	                            //table name parts:
	                            #tempTableNameParts := BYTE_TO_USINT(IN := #tdsTelegramArray[#tempTableNameByteCounter]);
	                            #tempTableNameByteCounter += 1;
	                            #tempTableNameTotalLength := 1;
	                            
	                            IF (#tempTableNameParts > 0) THEN
	                              
	                              //iteration throuh all table name parts
	                              FOR #tempTableNamePartCounter := 1 TO #tempTableNameParts DO
	                                //first two Bytes give table name length
	                                #tempTableNameLength := WORD_TO_UINT("LGF_MergeBytesToWord"(byte0 := #tdsTelegramArray[#tempTableNameByteCounter], byte1 := #tdsTelegramArray[#tempTableNameByteCounter + 1]));
	                                
	                                //each 1 character length takes 2 Bytes
	                                #tempTableNameByteCounter += 2 + 2 * UDINT_TO_DINT(#tempTableNameLength);
	                                #tempTableNameTotalLength += 2 + 2 * #tempTableNameLength;
	                                
	                              END_FOR;
	                              
	                            END_IF;
	                          END_REGION Table Names
	                          
	                          #tempTypeLengthOffset := #tempColumnSizeFieldSize + #TDS_COLUMNMETADATA_COLLATELENGTH + UDINT_TO_USINT(#tempTableNameTotalLength);
	                          
	                        36..47://UNIQUE, VARBINARY, INTN, VARCHAR, BINARY, CHAR
	                          #tempColumnSizeFieldSize := #TDS_COLUMN_SIZEFIELDSIZE_1;
	                          #tempTypeLengthOffset := #tempColumnSizeFieldSize;
	                        48..67:
	                          #tempColumnSizeFieldSize := #TDS_COLUMN_SIZEFIELDSIZE_0;
	                          #tempTypeLengthOffset := #tempColumnSizeFieldSize;
	                          CASE #columns[#tempColumnLoopCounter].columnType OF
	                            48://INT1
	                              #tempColumnSize := #TDS_COLUMN_SIZE_1;
	                            50://BIT
	                              #tempColumnSize := #TDS_COLUMN_SIZE_1;
	                            52://INT2
	                              #tempColumnSize := #TDS_COLUMN_SIZE_2;
	                            56://INT4
	                              #tempColumnSize := #TDS_COLUMN_SIZE_4;
	                            58://DATETIME4
	                              #tempColumnSize := #TDS_COLUMN_SIZE_4;
	                            59://REAL
	                              #tempColumnSize := #TDS_COLUMN_SIZE_4;
	                            60://MONEY
	                              #tempColumnSize := #TDS_COLUMN_SIZE_8;
	                            61://DATETIME
	                              #tempColumnSize := #TDS_COLUMN_SIZE_8;
	                            62://FLT8
	                              #tempColumnSize := #TDS_COLUMN_SIZE_8;
	                            64://SINT1
	                              #tempColumnSize := #TDS_COLUMN_SIZE_1;
	                            65://UINT2
	                              #tempColumnSize := #TDS_COLUMN_SIZE_2;
	                            66://UINT4
	                              #tempColumnSize := #TDS_COLUMN_SIZE_4;
	                            67://UINT8
	                              #tempColumnSize := #TDS_COLUMN_SIZE_8;
	                            ELSE
	                              #status := #ERR_COLUMNS_TYPENOTDEFINED;
	                              #statError := TRUE;
	                              GOTO END;
	                          END_CASE;
	                        98://VARIANT
	                          #tempColumnSizeFieldSize := #TDS_COLUMN_SIZEFIELDSIZE_4;
	                          #tempTypeLengthOffset := #tempColumnSizeFieldSize;
	                        #TDS_COLUMNTYPE_NTEXT://99 - NTEXT
	                          #tempColumnSizeFieldSize := #TDS_COLUMN_SIZEFIELDSIZE_4;
	                          
	                          REGION Table Names
	                            #tempTableNameByteCounter := #tempByteAddressCounter + #TDS_COLUMNMETADATA_COLUMNTYPEPOSOFFSET + 1 + #tempColumnSizeFieldSize + #TDS_COLUMNMETADATA_COLLATELENGTH;
	                            
	                            //table name parts:
	                            #tempTableNameParts := BYTE_TO_USINT(IN := #tdsTelegramArray[#tempTableNameByteCounter]);
	                            #tempTableNameByteCounter += 1;
	                            #tempTableNameTotalLength := 1;
	                            
	                            IF (#tempTableNameParts > 0) THEN
	                              
	                              //iteration throuh all table name parts
	                              FOR #tempTableNamePartCounter := 1 TO #tempTableNameParts DO
	                                //first two Bytes give table name length
	                                #tempTableNameLength := WORD_TO_UINT("LGF_MergeBytesToWord"(byte0 := #tdsTelegramArray[#tempTableNameByteCounter], byte1 := #tdsTelegramArray[#tempTableNameByteCounter + 1]));
	                                
	                                //each 1 character length takes 2 Bytes
	                                #tempTableNameByteCounter += 2 + 2 * UDINT_TO_DINT(#tempTableNameLength);
	                                #tempTableNameTotalLength += 2 + 2 * #tempTableNameLength;
	                                
	                              END_FOR;
	                              
	                            END_IF;
	                          END_REGION Table Names
	                          
	                          #tempTypeLengthOffset := #tempColumnSizeFieldSize + #TDS_COLUMNMETADATA_COLLATELENGTH + UDINT_TO_USINT(#tempTableNameTotalLength);
	                        103..104://NVARCHAR, BITN
	                          #tempColumnSizeFieldSize := #TDS_COLUMN_SIZEFIELDSIZE_1;
	                          #tempTypeLengthOffset := #tempColumnSizeFieldSize;
	                        106..108://DECIMAL, NUMERIC
	                          #tempColumnSizeFieldSize := #TDS_COLUMN_SIZEFIELDSIZE_1;
	                          #tempTypeLengthOffset := #tempColumnSizeFieldSize + 2;//type length size + precision + scale
	                        109..111://FLTN, MONEYN, DATETIMN
	                          #tempColumnSizeFieldSize := #TDS_COLUMN_SIZEFIELDSIZE_1;
	                          #tempTypeLengthOffset := #tempColumnSizeFieldSize;
	                        122://MONEY4
	                          #tempColumnSizeFieldSize := #TDS_COLUMN_SIZEFIELDSIZE_0;
	                          #tempTypeLengthOffset := #tempColumnSizeFieldSize;
	                          #tempColumnSize := #TDS_COLUMN_SIZE_4;
	                        127://INT8
	                          #tempColumnSizeFieldSize := #TDS_COLUMN_SIZEFIELDSIZE_0;
	                          #tempTypeLengthOffset := #tempColumnSizeFieldSize;
	                          #tempColumnSize := #TDS_COLUMN_SIZE_8;
	                        165://VARBINARY
	                          #tempColumnSizeFieldSize := #TDS_COLUMN_SIZEFIELDSIZE_2;
	                          #tempTypeLengthOffset := #tempColumnSizeFieldSize;
	                        167://VARCHAR
	                          #tempColumnSizeFieldSize := #TDS_COLUMN_SIZEFIELDSIZE_2;
	                          #tempTypeLengthOffset := #tempColumnSizeFieldSize + #TDS_COLUMNMETADATA_COLLATELENGTH;
	                        173://BINARY
	                          #tempColumnSizeFieldSize := #TDS_COLUMN_SIZEFIELDSIZE_2;
	                          #tempTypeLengthOffset := #tempColumnSizeFieldSize;
	                        175://CHAR
	                          #tempColumnSizeFieldSize := #TDS_COLUMN_SIZEFIELDSIZE_2;
	                          #tempTypeLengthOffset := #tempColumnSizeFieldSize + #TDS_COLUMNMETADATA_COLLATELENGTH;
	                        225://LONGBINARY
	                          #tempColumnSizeFieldSize := #TDS_COLUMN_SIZEFIELDSIZE_4;
	                          #tempTypeLengthOffset := #tempColumnSizeFieldSize;
	                        231..239://NVARCHAR, NCHAR
	                          #tempColumnSizeFieldSize := #TDS_COLUMN_SIZEFIELDSIZE_2;
	                          #tempTypeLengthOffset := #tempColumnSizeFieldSize + #TDS_COLUMNMETADATA_COLLATELENGTH;
	                        ELSE
	                          #status := #ERR_COLUMNS_TYPENOTDEFINED;
	                          #statError := TRUE;
	                          GOTO END;
	                      END_CASE;
	                      
	                      //write column size field size to current column collection item
	                      #columns[#tempColumnLoopCounter].columnSizeFieldSize := UINT_TO_USINT(#tempColumnSizeFieldSize);
	                      
	                      //read column size from the size field (if the size field size was > 0)
	                      IF (#tempColumnSizeFieldSize > #TDS_COLUMN_SIZEFIELDSIZE_0) THEN
	                        CASE #tempColumnSizeFieldSize OF
	                          #TDS_COLUMN_SIZEFIELDSIZE_1:
	                            //extract column size from the given field of a size of 1 byte
	                            #tempColumnSize := BYTE_TO_UDINT(#tdsTelegramArray[#tempByteAddressCounter + #TDS_COLUMNMETADATA_COLUMNTYPEPOSOFFSET + 1]);
	                          #TDS_COLUMN_SIZEFIELDSIZE_2:
	                            //extract column size from the given field of a size of 2 byte
	                            #tempColumnSize := DWORD_TO_UDINT("LGF_MergeBytesToDWord"(byte0 := #tdsTelegramArray[#tempByteAddressCounter + #TDS_COLUMNMETADATA_COLUMNTYPEPOSOFFSET + 1], byte1 := #tdsTelegramArray[#tempByteAddressCounter + #TDS_COLUMNMETADATA_COLUMNTYPEPOSOFFSET + 2], byte2 := #BYTE_EMPTY, byte3 := #BYTE_EMPTY));
	                          #TDS_COLUMN_SIZEFIELDSIZE_4:
	                            //extract column size from the given field of a size of 4 byte
	                            #tempColumnSize := DWORD_TO_UDINT("LGF_MergeBytesToDWord"(byte0 := #tdsTelegramArray[#tempByteAddressCounter + #TDS_COLUMNMETADATA_COLUMNTYPEPOSOFFSET + 1], byte1 := #tdsTelegramArray[#tempByteAddressCounter + #TDS_COLUMNMETADATA_COLUMNTYPEPOSOFFSET + 2], byte2 := #tdsTelegramArray[#tempByteAddressCounter + #TDS_COLUMNMETADATA_COLUMNTYPEPOSOFFSET + 3], byte3 := #tdsTelegramArray[#tempByteAddressCounter + #TDS_COLUMNMETADATA_COLUMNTYPEPOSOFFSET + 4]));
	                        END_CASE;
	                      END_IF;
	                      
	                      //finally write column size to current column collection item
	                      #columns[#tempColumnLoopCounter].columnSize := #tempColumnSize;
	                      
	                      //check column size to be a reasonable value
	                      IF (#tempColumnSize <= 0) THEN
	                        //cloumn size is negative
	                        #status := #ERR_COLUMNS_SIZENOTDEFINED;
	                        #statError := TRUE;
	                        GOTO END;
	                      ELSIF ((#tempColumnSize > (UPPER_BOUND(ARR := #tdsTelegramArray, DIM := 1) - #tempByteAddressCounter))) THEN
	                        //column size is larger than the rest of the data array and would cause this user program to crash
	                        
	                        //exclude special values from this check, e.g. a max. value 16#7FFFFFFE has a special meaning of NULL
	                        IF NOT (#tempColumnSizeFieldSize = #TDS_COLUMN_SIZE_4 AND #tempColumnSize >= #TDS_COLUMN_SIZE_4_MAXVALUE) AND NOT (#columns[#tempColumnLoopCounter].columnType = #TDS_COLUMNTYPE_VARIANT AND #tempColumnSize >= #TDS_COLUMNTYPE_VARIANT_MAXLENGTH) THEN
	                          #status := #ERR_TYPESIZEINCORRECT;
	                          #statError := TRUE;
	                          GOTO END;
	                        END_IF;
	                      END_IF;
	                      
	                    END_REGION type length
	                    
	                    REGION column name
	                      //get the length of the column name from next byte
	                      #columns[#tempColumnLoopCounter].columnNameLength := BYTE_TO_INT(IN := #tdsTelegramArray[#tempByteAddressCounter + #TDS_COLUMNMETADATA_COLUMNNAMEPOSOFFSET + #tempTypeLengthOffset]);
	                      
	                      //move bytes to temporary array and then call function for transformation of Bytes to String
	                      MOVE_BLK(IN    := #tdsTelegramArray[#tempByteAddressCounter + #TDS_COLUMNMETADATA_COLUMNNAMEPOSOFFSET + 1 + #tempTypeLengthOffset],
	                               COUNT := 2 * INT_TO_UDINT(#columns[#tempColumnLoopCounter].columnNameLength),
	                               OUT   => #tempByteCharArray[0]);
	                      
	                      #columns[#tempColumnLoopCounter].columnName := "LSql_BytesToString"(columnType := 0, byteArray := #tempByteCharArray, numberOfBytes := 2 * INT_TO_UINT(#columns[#tempColumnLoopCounter].columnNameLength));
	                    END_REGION column name
	                    
	                    //increment byte address counter by the size/length of all values that haven been used for the current column
	                    #tempByteAddressCounter += INT_TO_USINT(#TDS_COLUMNMETADATA_COLUMNNAMEPOS + USINT_TO_INT(#tempTypeLengthOffset) + 2 * #columns[#tempColumnLoopCounter].columnNameLength);
	                    
	                    //check whether last column has been analyzed
	                    IF (#tempColumnLoopCounter >= #columnCount - 1) THEN
	                      #statMetaDataAvailable := true;
	                    END_IF;
	                    
	                  ELSE
	                    //the upper slots of the column array will not be filled with received columns anymore
	                    //loop execiution can be ended
	                    //the number of valid columns is explicitly given as output parameter
	                    EXIT;
	                    
	                  END_IF;
	                  
	                END_FOR;
	                
	              END_REGION #columns
	              
	            END_REGION Token - ColumnMetaData
	            
	          #TDS_TOKENROW_TOKENTYPE:
	            REGION Token - Row
	              
	              //check that ColumnMetaData have been anaylzed before accessing the row tokens
	              IF #statMetaDataAvailable THEN
	                
	                // set rowDataStart at first passing
	                IF (#rowDataStart <= 0) THEN
	                  #rowDataStart := DINT_TO_UINT(#tempByteAddressCounter);
	                END_IF;
	                
	                //increment for token type 'D1'
	                #tempByteAddressCounter += #TDS_TOKEN_TYPEFIELDLENGTH;
	                #rowDataLength += #TDS_TOKEN_TYPEFIELDLENGTH;
	                
	                //loop through the known colum meta data
	                FOR #tempColumnLoopCounter := 0 TO #columnCount - 1 BY 1
	                DO
	                  #tempColumnLength := #columns[#tempColumnLoopCounter].columnSize;
	                  
	                  //datatypes TEXT and NTEXT bring additional Data: 'Data Textptr Len', 'Data Textptr' and 'Data Text timestamp'
	                  IF (#columns[#tempColumnLoopCounter].columnType = #TDS_COLUMNTYPE_TEXT OR #columns[#tempColumnLoopCounter].columnType = #TDS_COLUMNTYPE_NTEXT) THEN
	                    #tempRowDataTextptrLen := BYTE_TO_USINT(#tdsTelegramArray[#tempByteAddressCounter]);
	                    
	                    //increment counter by lengths of the additional fields
	                    #tempRowDataTextTotalLength := 1 + #tempRowDataTextptrLen + #TDS_TOKENROW_DATATEXTTIMESTAMP_LENGTH;
	                    #tempByteAddressCounter += UDINT_TO_DINT(#tempRowDataTextTotalLength);
	                  ELSE
	                    #tempRowDataTextTotalLength := 0;
	                  END_IF;
	                  
	                  //check if there is a field for the column size
	                  IF (#columns[#tempColumnLoopCounter].columnSizeFieldSize > 0) THEN
	                    #tempColumnLength := 0;
	                    
	                    //read out the actual length
	                    CASE #columns[#tempColumnLoopCounter].columnSizeFieldSize OF
	                      #TDS_COLUMN_SIZEFIELDSIZE_1:
	                        #tempColumnLength := DWORD_TO_UDINT("LGF_MergeBytesToDWord"(byte0 := #tdsTelegramArray[#tempByteAddressCounter], byte1 := #BYTE_EMPTY, byte2 := #BYTE_EMPTY, byte3 := #BYTE_EMPTY));
	                      #TDS_COLUMN_SIZEFIELDSIZE_2:
	                        #tempColumnLength := DWORD_TO_UDINT("LGF_MergeBytesToDWord"(byte0 := #tdsTelegramArray[#tempByteAddressCounter], byte1 := #tdsTelegramArray[#tempByteAddressCounter + 1], byte2 := #BYTE_EMPTY, byte3 := #BYTE_EMPTY));
	                      #TDS_COLUMN_SIZEFIELDSIZE_4:
	                        #tempColumnLength := DWORD_TO_UDINT("LGF_MergeBytesToDWord"(byte0 := #tdsTelegramArray[#tempByteAddressCounter], byte1 := #tdsTelegramArray[#tempByteAddressCounter + 1], byte2 := #tdsTelegramArray[#tempByteAddressCounter + 2], byte3 := #tdsTelegramArray[#tempByteAddressCounter + 3]));
	                      ELSE
	                        #tempColumnLength := #columns[#tempColumnLoopCounter].columnSize;
	                    END_CASE;
	                    
	                    //check if the value is out of range
	                    IF (#tempColumnLength < 0 OR #tempColumnLength > #columns[#tempColumnLoopCounter].columnSize) THEN
	                      #tempColumnLength := 0;
	                    END_IF;
	                  END_IF;
	                  
	                  //check wehther the given length of the value exceeds the byte array boundaries and would cause a program crash
	                  IF (#tempColumnLength > UPPER_BOUND(ARR := #tdsTelegramArray, DIM := 1) - #tempByteAddressCounter) THEN
	                    #status := #ERR_TYPESIZEINCORRECT;
	                    #statBusy := FALSE;
	                    #statError := TRUE;
	                    GOTO END;
	                  ELSE
	                    //increment counter by length field and length value
	                    #tempByteAddressCounter += #columns[#tempColumnLoopCounter].columnSizeFieldSize + UDINT_TO_DINT(#tempColumnLength);
	                    #rowDataLength += #columns[#tempColumnLoopCounter].columnSizeFieldSize + #tempColumnLength;
	                  END_IF;
	                  
	                END_FOR;
	                
	                //set output that telegram contains rows and they are available
	                #statRowsAvailable := TRUE;
	                
	              ELSE
	                //there are no ColumnMetaData information to be used for analyzing the rows
	                #status := #ERR_TOKENROW_NOMETADATA;
	                #statBusy := FALSE;
	                #statError := TRUE;
	                GOTO END;
	              END_IF;
	              
	            END_REGION Token - Row
	            
	          #TDS_TOKENORDER_TOKENTYPE:
	            REGION Token - Order
	              //total token length is given in the token itself
	              #tempTokenLength := WORD_TO_UINT("LGF_MergeBytesToWord"(byte0 := #tdsTelegramArray[#tempByteAddressCounter + 1], byte1 := #tdsTelegramArray[#tempByteAddressCounter + 2]));
	              
	              //increment counter by length field and length value
	              #tempByteAddressCounter += #TDS_TOKEN_TYPEFIELDLENGTH + #TDS_TOKEN_LENGTHFIELDLENGTH + #tempTokenLength;
	            END_REGION Token - Order
	            
	          #TDS_TOKENERROR_TOKENTYPE:
	            REGION Token - Error
	              #status := #ERR_TOKENERROR;
	              #statError := TRUE;
	              
	              REGION Token Length
	                #errorToken.TokenLength := WORD_TO_UINT("LGF_MergeBytesToWord"(byte0 := #tdsTelegramArray[#tempByteAddressCounter + #TDS_TOKENERROR_TOKENLENGTHPOS], byte1 := #tdsTelegramArray[#tempByteAddressCounter + #TDS_TOKENERROR_TOKENLENGTHPOS + 1]));
	              END_REGION Token Length
	              
	              REGION SQL Error Number
	                #errorToken.SQLErrorNumber := DWORD_TO_UDINT("LGF_MergeBytesToDWord"(byte3 := #tdsTelegramArray[#tempByteAddressCounter + #TDS_TOKENERROR_SQLERRORNUMBERPOS + 3], byte2 := #tdsTelegramArray[#tempByteAddressCounter + #TDS_TOKENERROR_SQLERRORNUMBERPOS + 2], byte1 := #tdsTelegramArray[#tempByteAddressCounter + #TDS_TOKENERROR_SQLERRORNUMBERPOS + 1], byte0 := #tdsTelegramArray[#tempByteAddressCounter + #TDS_TOKENERROR_SQLERRORNUMBERPOS]));
	              END_REGION SQL Error Number
	              
	              REGION State and Class
	                #errorToken.State := #tdsTelegramArray[#tempByteAddressCounter + #TDS_TOKENERROR_STATEPOS];
	                #errorToken.Class := BYTE_TO_USINT(#tdsTelegramArray[#tempByteAddressCounter + #TDS_TOKENERROR_CLASSPOS]);
	              END_REGION State and Class
	              
	              REGION Error Message
	                //field 'ErrorMessageLength'
	                #tempByteAddressCounter += #TDS_TOKENERROR_ERRORMESSAGELENGTHPOS;
	                #errorToken.ErrorMessageLength := WORD_TO_UINT("LGF_MergeBytesToWord"(byte0 := #tdsTelegramArray[#tempByteAddressCounter], byte1 := #tdsTelegramArray[#tempByteAddressCounter + 1]));
	                
	                //field "ErrorMessage' as String
	                //move bytes to temporary array and then call function for transformation of Bytes to String
	                MOVE_BLK(IN    := #tdsTelegramArray[#tempByteAddressCounter + #TDS_TOKENERROR_ERRORMESSAGELENGTHLENGTH],
	                         COUNT := 2 * #errorToken.ErrorMessageLength,
	                         OUT   => #tempByteCharArray[0]);
	                
	                #errorToken.ErrorMessage := "LSql_BytesToString"(columnType := 0, byteArray := #tempByteCharArray, numberOfBytes := 2 * #errorToken.ErrorMessageLength);
	                
	                //increment address counter by length field and dynamic value length
	                #tempByteAddressCounter += #TDS_TOKENERROR_ERRORMESSAGELENGTHLENGTH + (#errorToken.ErrorMessageLength * 2);
	              END_REGION Error Message
	              
	              REGION Server Name
	                //field "ServerNameLength'
	                #errorToken.ServerNameLength := BYTE_TO_USINT(#tdsTelegramArray[#tempByteAddressCounter]);
	                
	                //field "ServerName' as String
	                //move bytes to temporary array and then call function for transformation of Bytes to String
	                MOVE_BLK(IN    := #tdsTelegramArray[#tempByteAddressCounter + #TDS_TOKENERROR_SERVERNAMELENGTHLENGTH],
	                         COUNT := 2 * #errorToken.ServerNameLength,
	                         OUT   => #tempByteCharArray[0]);
	                
	                #errorToken.ServerName := "LSql_BytesToString"(columnType := 0, byteArray := #tempByteCharArray, numberOfBytes := 2 * #errorToken.ServerNameLength);
	                
	                //increment address counter by length field and dynamic value length
	                #tempByteAddressCounter += #TDS_TOKENERROR_SERVERNAMELENGTHLENGTH + (#errorToken.ServerNameLength * 2);
	              END_REGION Server Name
	              
	              REGION Procedure Name
	                //field 'ProcNameLength'
	                #errorToken.ProcNameLength := BYTE_TO_USINT(#tdsTelegramArray[#tempByteAddressCounter]);
	                
	                //field 'ProcName' as String
	                //move bytes to temporary array and then call function for transformation of Bytes to String
	                MOVE_BLK(IN    := #tdsTelegramArray[#tempByteAddressCounter + #TDS_TOKENERROR_PROCNAMELENGTHLENGTH],
	                         COUNT := 2 * #errorToken.ProcNameLength,
	                         OUT   => #tempByteCharArray[0]);
	                
	                #errorToken.ProcName := "LSql_BytesToString"(columnType := 0, byteArray := #tempByteCharArray, numberOfBytes := 2 * #errorToken.ProcNameLength);
	                
	                //increment address counter by length field and dynamic value length
	                #tempByteAddressCounter += + #TDS_TOKENERROR_PROCNAMELENGTHLENGTH + (#errorToken.ProcNameLength * 2);
	              END_REGION Procedure Name
	              
	              REGION Line Number
	                #errorToken.LineNumber := DWORD_TO_UDINT("LGF_MergeBytesToDWord"(byte0 := #tdsTelegramArray[#tempByteAddressCounter], byte1 := #tdsTelegramArray[#tempByteAddressCounter + 1], byte2 := #tdsTelegramArray[#tempByteAddressCounter + 2], byte3 := #tdsTelegramArray[#tempByteAddressCounter + 3]));
	                
	                //increment counter by field length
	                #tempByteAddressCounter += #TDS_TOKENERROR_LINENUMBERLENGTH;
	              END_REGION Line Number
	              
	            END_REGION Token - Error
	            
	          #TDS_TOKENDONE_TOKENTYPE:
	            REGION Token - Done
	              //next two byte are status field
	              #tempTokenEndStatus := WORD_TO_UINT("LGF_MergeBytesToWord"(byte0 := #tdsTelegramArray[#tempByteAddressCounter + 1], byte1 := #tdsTelegramArray[#tempByteAddressCounter + 2]));
	              
	              CASE #tempTokenEndStatus OF
	                #TDS_TOKENDONE_STATUSDONEFINAL:
	                  //status case not handled in this application example
	                  ;
	                #TDS_TOKENDONE_STATUSDONEMORE:
	                  //status case not handled in this application example
	                  ;
	                #TDS_TOKENDONE_STATUSDONEERROR:
	                  //status case not handled in this application example
	                  ;
	                #TDS_TOKENDONE_STATUSDONEINXACT:
	                  //status case not handled in this application example
	                  ;
	                #TDS_TOKENDONE_STATUSDONECOUNT:
	                  //tokenDone contains the number of tokenRows
	                  #rowCount := DWORD_TO_UDINT("LGF_MergeBytesToDWord"(byte0 := #tdsTelegramArray[#tempByteAddressCounter + #TDS_TOKENDONE_STATUSDONE_ROWCOUNTPOS], byte1 := #tdsTelegramArray[#tempByteAddressCounter + #TDS_TOKENDONE_STATUSDONE_ROWCOUNTPOS + 1], byte2 := #tdsTelegramArray[#tempByteAddressCounter + #TDS_TOKENDONE_STATUSDONE_ROWCOUNTPOS + 2], byte3 := #tdsTelegramArray[#tempByteAddressCounter + #TDS_TOKENDONE_STATUSDONE_ROWCOUNTPOS + 3]));
	                #TDS_TOKENDONE_STATUSDONEATTN:
	                  //status case not handled in this application example
	                  ;
	                #TDS_TOKENDONE_STATUSDONESRVERROR:
	                  //status case not handled in this application example
	                  ;
	                ELSE
	                  //unknown or wrong status of Token Done
	                  #status := #ERR_TOKENDONE_UNKNOWNSTATUS;
	                  #statBusy := FALSE;
	                  #statError := TRUE;
	                  //reset rowCount output value
	                  #rowCount := 0;
	                  GOTO END;
	              END_CASE;
	              
	              //increment counter by fixed length value
	              #tempByteAddressCounter += #TDS_TOKENDONE_LENGTH;
	            END_REGION Token - Done
	            
	          #TDS_TOKENDONEINPROC_TOKENTYPE:
	            REGION Token - DoneInProc
	              //tokenDone contains the number of tokenRows
	              #rowCount := DWORD_TO_UDINT("LGF_MergeBytesToDWord"(byte0 := #tdsTelegramArray[#tempByteAddressCounter + #TDS_TOKENDONEINPROC_ROWCOUNTPOS], byte1 := #tdsTelegramArray[#tempByteAddressCounter + #TDS_TOKENDONEINPROC_ROWCOUNTPOS + 1], byte2 := #tdsTelegramArray[#tempByteAddressCounter + #TDS_TOKENDONEINPROC_ROWCOUNTPOS + 2], byte3 := #tdsTelegramArray[#tempByteAddressCounter + #TDS_TOKENDONEINPROC_ROWCOUNTPOS + 3]));
	              
	              //increment counter by fixed length value
	              #tempByteAddressCounter += #TDS_TOKENDONEINPROC_LENGTH;
	            END_REGION Token - DoneInProc
	            
	          #TDS_TOKENRETURNSTATUS_TOKENTYPE:
	            REGION Token - ReturnStatus
	              //increment counter by fixed length value
	              #tempByteAddressCounter += #TDS_TOKENRETURNSTATUS_LENGTH;
	            END_REGION Token - ReturnStatus
	            
	          #TDS_TOKENDONEPROC_TOKENTYPE:
	            REGION Token - DoneProc
	              //increment counter by fixed length value
	              #tempByteAddressCounter += #TDS_TOKENDONEPROC_LENGTH;
	            END_REGION Token - DoneProc
	            
	          #TDS_TOKENINFO_TOKENTYPE:
	            REGION Token - Info
	              #tempTokenLength := WORD_TO_UINT("LGF_MergeBytesToWord"(byte0 := #tdsTelegramArray[#tempByteAddressCounter + 1], byte1 := #tdsTelegramArray[#tempByteAddressCounter + 2]));
	              
	              //increment counter by length field and length value
	              #tempByteAddressCounter += #TDS_TOKEN_TYPEFIELDLENGTH + #TDS_TOKEN_LENGTHFIELDLENGTH + #tempTokenLength;
	            END_REGION Token - Info
	            
	          #TDS_TOKENENVCHANGE_TOKENTYPE:
	            REGION Token - EnvChange
	              #tempTokenLength := WORD_TO_UINT("LGF_MergeBytesToWord"(byte0 := #tdsTelegramArray[#tempByteAddressCounter + 1], byte1 := #tdsTelegramArray[#tempByteAddressCounter + 2]));
	              
	              //increment counter by length field and length value
	              #tempByteAddressCounter += #TDS_TOKEN_TYPEFIELDLENGTH + #TDS_TOKEN_LENGTHFIELDLENGTH + #tempTokenLength;
	            END_REGION Token - EnvChange
	            
	          ELSE
	            REGION Unknown token type
	              //the token type is unknown, the iteration can not go on because there is no length information about that next token
	              #status := #ERR_UNKNOWNTOKEN;
	              #statBusy := FALSE;
	              #statError := TRUE;
	              GOTO END;
	            END_REGION Unknown token type
	        END_CASE;
	        
	      END_WHILE;
	      
	    END_REGION Tokens
	    
	    //reconfirm that the number of analyzed bytes is exactly matching the total telegram length:
	    IF (#tempByteAddressCounter = #tdsHeader.length) THEN
	      //operation completed
	      #statBusy := FALSE;
	      #statDone := TRUE;
	    ELSE
	      #status := #ERR_LENGTHINCORRECT;
	      #statBusy := FALSE;
	      #statError := TRUE;
	      GOTO END;
	    END_IF;
	    
	  END_REGION Execution
	  
	ELSIF NOT #execute THEN
	  REGION Idle state
	    //not executing, reset output values
	    #statDone := FALSE;
	    #statBusy := FALSE;
	    #statError := FALSE;
	    #status := #ERR_NOERROR;
	    #statRowsAvailable := FALSE;
	    #statMetaDataAvailable := FALSE;
	    #rowCount := 0;
	  END_REGION Idle state
	END_IF;
	
	END:
	REGION WRITE OUTPUTS
	  //finally write static values to outputs
	  #metaDataAndRowsAvailable := #statRowsAvailable AND #statMetaDataAvailable AND #statDone;
	  #error := #statError;
	  #busy := #statBusy;
	  #done := #statDone;
	END_REGION WRITE OUTPUTS
END_FUNCTION_BLOCK

FUNCTION_BLOCK "DeserializeRows"
TITLE = DeserializeRows
{ S7_Optimized_Access := 'TRUE' }
AUTHOR : 'SIEMENS AG'
VERSION : 3.0
//FB for using the ColumnMetaData and rowCount information in order to transform the row payload of Tabular Data Stream byte array into tokenRows of use case specific structure
   VAR_INPUT 
      columnCount { ExternalAccessible := 'False'; ExternalVisible := 'False'; ExternalWritable := 'False'} : UInt;   // numberof received columns
      columns { ExternalAccessible := 'False'; ExternalVisible := 'False'; ExternalWritable := 'False'} : Array[0.."LSQL_NUMBER_OF_COLUMNS_MAX"] of "LSql_typeColumn";
      rowCount { ExternalAccessible := 'False'; ExternalVisible := 'False'; ExternalWritable := 'False'} : UDInt;   // number of received rows
      rowDataStart { ExternalAccessible := 'False'; ExternalVisible := 'False'; ExternalWritable := 'False'} : UInt;   // start byte address of row data area
      rowDataLength { ExternalAccessible := 'False'; ExternalVisible := 'False'; ExternalWritable := 'False'} : UDInt;   // byte length of row data area
      numberOfRowsPerCycle { ExternalAccessible := 'False'; ExternalVisible := 'False'; ExternalWritable := 'False'} : USInt;   // number of rows to be deserialized per cycle
      execute { ExternalAccessible := 'False'; ExternalVisible := 'False'; ExternalWritable := 'False'} : Bool;   // bit flag for triggering execution
   END_VAR

   VAR_OUTPUT 
      busy { ExternalAccessible := 'False'; ExternalVisible := 'False'; ExternalWritable := 'False'} : Bool := FALSE;   // TRUE = execution is running
      done { ExternalAccessible := 'False'; ExternalVisible := 'False'; ExternalWritable := 'False'} : Bool := FALSE;   // TRUE = execution is done
      error { ExternalAccessible := 'False'; ExternalVisible := 'False'; ExternalWritable := 'False'} : Bool := FALSE;   // TRUE = execution has error
      warning { ExternalAccessible := 'False'; ExternalVisible := 'False'; ExternalWritable := 'False'} : Bool := FALSE;   // TRUE = execution has warning, e.g. a column field is not used by program code
      rowOverflow { ExternalAccessible := 'False'; ExternalVisible := 'False'; ExternalWritable := 'False'} : Bool := FALSE;   // TRUE = more rows from TDS than items in UDT array
      status { ExternalAccessible := 'False'; ExternalVisible := 'False'; ExternalWritable := 'False'} : Word := 16#0;   // status code
   END_VAR

   VAR_IN_OUT 
      tdsTelegramArray : Array[*] of Byte;   // array of Bytes for row data
      rows : Array[*] of "typeTokenRow";
   END_VAR

   VAR 
      statRowOverflow { ExternalAccessible := 'False'; ExternalVisible := 'False'; ExternalWritable := 'False'} : Bool;   // static value for output 'rowOverflow'
      statBusy { ExternalAccessible := 'False'; ExternalVisible := 'False'; ExternalWritable := 'False'} : Bool;   // static value for output 'busy'
      statDone { ExternalAccessible := 'False'; ExternalVisible := 'False'; ExternalWritable := 'False'} : Bool;   // static value for output 'done'
      statError { ExternalAccessible := 'False'; ExternalVisible := 'False'; ExternalWritable := 'False'} : Bool;   // static value for output 'error'
      statWarning { ExternalAccessible := 'False'; ExternalVisible := 'False'; ExternalWritable := 'False'} : Bool;   // static value for output 'warning'
      statStatus { ExternalAccessible := 'False'; ExternalVisible := 'False'; ExternalWritable := 'False'} : Word;   // static value for output 'status'
      statRowsDeserialized { ExternalAccessible := 'False'; ExternalVisible := 'False'; ExternalWritable := 'False'} : UDInt;   // comulative counter of deserialized rows
      statByteAddressCounter { ExternalAccessible := 'False'; ExternalVisible := 'False'; ExternalWritable := 'False'} : DInt;   // comulative byte address in row data array
   END_VAR

   VAR_TEMP 
      tempRowLoopCounter : DInt;   // temp counter for row iteration
      tempRowLoopCounterUpper : DInt;   // upper bound of counter for row iteration
      tempColumnLoopCounter : UInt;   // temp counter for column iteration
      tempByteCharArray : Array[0..507] of Byte;   // temporary array of Byte to be transformed to String
      tempTokenRowsUpperBound : DInt;   // upper bound of tokenRows array
      tempTokenRowsLowerBound : DInt;   // lower bound of tokenRows array
      tempDWord : DWord;   // temp DWord for datatype conversion
      tempValueLength : UDInt;   // actual length of the value in a row token
      tempRowDataTextptrLen : USInt;   // length of additional field 'Textptr' in Row token
      tempRowDataTextTotalLength : UDInt;   // total length of additional fields 'Text' in Row data
   END_VAR

   VAR CONSTANT 
      BYTE_EMPTY : Byte := 16#0;   // empty Byte
      TDS_TOKENROW_COLUMNTYPE_TEXT : UInt := 35;   // identifier of SQL column tpye 'TEXT'
      TDS_TOKENROW_COLUMNTYPE_NTEXT : UInt := 99;   // identifier of SQL column type 'NTEXT'
      TDS_TOKENROW_DATATEXTTIMESTAMP_LENGTH : USInt := 8;   // length of field 'Data Text timesatmp'
      TDS_COLUMN_SIZEFIELDSIZE_0 : USInt := 0;   // size information is in field of size 0 byte
      TDS_COLUMN_SIZEFIELDSIZE_1 : USInt := 1;   // size information is in field of size 1 byte
      TDS_COLUMN_SIZEFIELDSIZE_2 : USInt := 2;   // size information is in field of size 2 byte
      TDS_COLUMN_SIZEFIELDSIZE_4 : USInt := 4;   // size information is in field of size 4 byte
      TDS_COLUMN_SIZEFIELDSIZE_8 : USInt := 8;   // size information is in field of size 8 byte
      ERR_NOERROR : Word := 16#0000;   // No Error.
      ERR_ROWARRAY_SIZENOTDEFINED : Word := 16#8601;   // Error: Row array size is not defined.
      ERR_ROWARRAY_SIZEINCORRECT : Word := 16#8602;   // Error: Row array size is incorrect.
      ERR_ROWDATA_LENGHTNOTDEFINED : Word := 16#8603;   // Error: Row data length is incorrect.
      ERR_COLUMNS_COUNTINCORRECT : Word := 16#8604;   // Error: Column count incorrect.
      ERR_COULMNS_COLUMNNOTEXISTING : Word := 16#8605;   // Error: At least one column name can not be handled.
   END_VAR


BEGIN
	REGION BLOCK INFO HEADER
	  //=============================================================================
	  // Siemens AG (c)Copyright (2022)
	  //-----------------------------------------------------------------------------
	  // Library:       SQL
	  // Target:        S7-1500 V2.9 / S7-1200 V4.5
	  // Engineering:   TIA Portal V17
	  // Restrictions:  no
	  // Requirements:  S7-1500 CPU / S7-1200 CPU
	  // Functionality: deserialize SELECT row data array into row tokens and transform values to use case data types
	  //-----------------------------------------------------------------------------
	  // Change log table:
	  // Version    Date         Expert in charge           Changes applied
	  // 01.00.00   31.01.2022   Siemens SUP Applications   initially added to project
	  // 01.00.01   29.09.2022   Siemens SUP Applications   - minor formatting changes
	  //                                                    - bugfix for datatypes TEXT and NTEXT; dynamic adaption to field lengths
	  //                                                    - deleted section for clearing unused rows because the number of valid rows is explicitly given
	  // 01.01.00   06.10.2022   Siemens SUP Applications   using FC 'Lsql_BytesToString' for transforming character-based bytes to String
	  //=============================================================================
	END_REGION
	
	IF (#execute AND NOT #statDone) THEN
	  #statBusy := TRUE;
	  
	  REGION check boundaries
	    //get upper and lower bound of Array[*]
	    #tempTokenRowsUpperBound := UPPER_BOUND(ARR := #rows, DIM := 1);
	    #tempTokenRowsLowerBound := LOWER_BOUND(ARR := #rows, DIM := 1);
	    //check for incorrect array boundaries or input values
	    IF #tempTokenRowsUpperBound - #tempTokenRowsLowerBound <= 0 THEN
	      #statStatus := #ERR_ROWARRAY_SIZENOTDEFINED;
	      #statError := TRUE;
	      GOTO END;
	    ELSIF #tempTokenRowsUpperBound <= 0 OR #tempTokenRowsLowerBound < 0 THEN
	      #statStatus := #ERR_ROWARRAY_SIZEINCORRECT;
	      #statError := TRUE;
	      GOTO END;
	    ELSIF #rowDataLength <= 0 THEN
	      #statStatus := #ERR_ROWDATA_LENGHTNOTDEFINED;
	      #statError := TRUE;
	      GOTO END;
	    ELSIF #columnCount <= 0 THEN
	      #statStatus := #ERR_COLUMNS_COUNTINCORRECT;
	      #statError := TRUE;
	      GOTO END;
	    END_IF;
	  END_REGION check boundaries  
	  
	  REGION check row overflow
	    //check if SELECT fills more rows than the number of available rows in tokenRow array
	    IF (#tempTokenRowsUpperBound - #tempTokenRowsLowerBound + 1 >= #rowCount) THEN
	      #statRowOverflow := FALSE;
	    ELSE
	      #statRowOverflow := TRUE;
	    END_IF;
	  END_REGION check row overflow
	  
	  REGION deserialize data
	    //start at lower array boundary on first call
	    IF (#statRowsDeserialized = 0) THEN
	      #statRowsDeserialized := DINT_TO_UDINT(#tempTokenRowsLowerBound);
	      #statByteAddressCounter := #rowDataStart;
	    END_IF;
	    
	    IF #numberOfRowsPerCycle <= 0 THEN
	      //number of rows to be deserialized per cycle is not set, so do all available rows at once
	      #tempRowLoopCounterUpper := #tempTokenRowsUpperBound;
	    ELSIF #tempTokenRowsLowerBound + UDINT_TO_DINT(#statRowsDeserialized) + #numberOfRowsPerCycle - 1 < #tempTokenRowsUpperBound THEN
	      //do the next batch of rows while upper bound of the array will not be reached yet
	      #tempRowLoopCounterUpper := #tempTokenRowsLowerBound + UDINT_TO_DINT(#statRowsDeserialized) + #numberOfRowsPerCycle - 1;
	    ELSE
	      //do the next batch of rows until the upper bound of the array will be reached
	      #tempRowLoopCounterUpper := #tempTokenRowsUpperBound;
	    END_IF;
	    
	    //iteration over rows of the row array
	    FOR #tempRowLoopCounter := (#tempTokenRowsLowerBound + UDINT_TO_DINT(#statRowsDeserialized)) TO #tempRowLoopCounterUpper BY 1
	    DO
	      //check if the array place will be occupied by a received row
	      IF #tempRowLoopCounter - #tempTokenRowsLowerBound < #rowCount THEN
	        
	        //each row token is started by one byte '0xd1' identifying it as a TokenType
	        #statByteAddressCounter += 1;
	        
	        //iteration over all columns given from ColumnMetaData
	        FOR #tempColumnLoopCounter := 0 TO #columnCount - 1 BY 1
	        DO
	          //datatypes TEXT and NTEXT bring additional Data: 'Data Textptr Len', 'Data Textptr' and 'Data Text timestamp'
	          IF (#columns[#tempColumnLoopCounter].columnType = #TDS_TOKENROW_COLUMNTYPE_TEXT OR #columns[#tempColumnLoopCounter].columnType = #TDS_TOKENROW_COLUMNTYPE_NTEXT) THEN
	            #tempRowDataTextptrLen := BYTE_TO_USINT(#tdsTelegramArray[#statByteAddressCounter]);
	            
	            #tempRowDataTextTotalLength := 1 + #tempRowDataTextptrLen + #TDS_TOKENROW_DATATEXTTIMESTAMP_LENGTH;
	            #statByteAddressCounter += UDINT_TO_DINT(#tempRowDataTextTotalLength);
	          ELSE
	            #tempRowDataTextTotalLength := 0;
	          END_IF;
	          
	          //check if there is a field for the column size
	          IF (#columns[#tempColumnLoopCounter].columnSizeFieldSize > 0) THEN
	            
	            #tempValueLength := 0;
	            
	            //read out the actual length
	            CASE #columns[#tempColumnLoopCounter].columnSizeFieldSize OF
	              #TDS_COLUMN_SIZEFIELDSIZE_1:
	                #tempValueLength := DWORD_TO_UDINT("LGF_MergeBytesToDWord"(byte0 := #tdsTelegramArray[#statByteAddressCounter], byte1 := #BYTE_EMPTY, byte2 := #BYTE_EMPTY, byte3 := #BYTE_EMPTY));
	              #TDS_COLUMN_SIZEFIELDSIZE_2:
	                #tempValueLength := DWORD_TO_UDINT("LGF_MergeBytesToDWord"(byte0 := #tdsTelegramArray[#statByteAddressCounter], byte1 := #tdsTelegramArray[#statByteAddressCounter + 1], byte2 := #BYTE_EMPTY, byte3 := #BYTE_EMPTY));
	              #TDS_COLUMN_SIZEFIELDSIZE_4:
	                #tempValueLength := DWORD_TO_UDINT("LGF_MergeBytesToDWord"(byte0 := #tdsTelegramArray[#statByteAddressCounter], byte1 := #tdsTelegramArray[#statByteAddressCounter + 1], byte2 := #tdsTelegramArray[#statByteAddressCounter + 2], byte3 := #tdsTelegramArray[#statByteAddressCounter + 3]));
	              ELSE
	                #tempValueLength := #columns[#tempColumnLoopCounter].columnSize;
	            END_CASE;
	            
	            IF (#tempValueLength < 0 OR #tempValueLength > #columns[#tempColumnLoopCounter].columnSize) THEN
	              #tempValueLength := 0;
	            END_IF;
	            
	          ELSE
	            #tempValueLength := #columns[#tempColumnLoopCounter].columnSize;
	          END_IF;
	          
	          //increment address counter
	          #statByteAddressCounter += #columns[#tempColumnLoopCounter].columnSizeFieldSize;
	          
	          REGION --> use case deserializaition
	            
	            //IF - ELSIF case selection on the columName
	            
	            IF #columns[#tempColumnLoopCounter].columnName = 'Pressure' THEN
	              REGION example INT
	                //merge next two BYTE to WORD and then convert to INT
	                #rows[#tempRowLoopCounter].Pressure := WORD_TO_INT("LGF_MergeBytesToWord"(byte0 := #tdsTelegramArray[#statByteAddressCounter], byte1 := #tdsTelegramArray[#statByteAddressCounter + 1]));
	            END_REGION example Int
	            
	            ELSIF #columns[#tempColumnLoopCounter].columnName = 'Temperature' THEN
	                REGION example INT2
	                    //merge next two BYTE to WORD and then convert to INT
	                    #rows[#tempRowLoopCounter].Temperature := WORD_TO_INT("LGF_MergeBytesToWord"(byte0 := #tdsTelegramArray[#statByteAddressCounter], byte1 := #tdsTelegramArray[#statByteAddressCounter + 1]));
	                END_REGION example Int2
	         (*     
	            ELSIF #columns[#tempColumnLoopCounter].columnName = 'Fresh' THEN
	             REGION example Bool
	                //convert BYTE to BOOL
	                #rows[#tempRowLoopCounter].Fresh := BYTE_TO_BOOL(#tdsTelegramArray[#statByteAddressCounter]);
	              END_REGION example Bool
	              
	            ELSIF #columns[#tempColumnLoopCounter].columnName = 'Color' THEN
	              REGION example String
	                //move Bytes to temporary array
	                MOVE_BLK(IN    := #tdsTelegramArray[#statByteAddressCounter],
	                         COUNT := UDINT_TO_UINT(#tempValueLength),
	                         OUT   => #tempByteCharArray[0]);
	                
	                //convert BYTE array to STRING
	                #rows[#tempRowLoopCounter].Temperature := "LSql_BytesToString"(columnType := #columns[#tempColumnLoopCounter].columnType, byteArray := #tempByteCharArray, numberOfBytes := UDINT_TO_UINT(#tempValueLength));
	              END_REGION example String
	              
	            ELSIF #columns[#tempColumnLoopCounter].columnName = 'Fruit' THEN
	              REGION example String
	                //move Bytes to temporary array
	                MOVE_BLK(IN    := #tdsTelegramArray[#statByteAddressCounter],
	                         COUNT := UDINT_TO_UINT(#tempValueLength),
	                         OUT   => #tempByteCharArray[0]);
	                
	                //convert BYTE array to STRING
	                #rows[#tempRowLoopCounter].Fruit := "LSql_BytesToString"(columnType := #columns[#tempColumnLoopCounter].columnType, byteArray := #tempByteCharArray, numberOfBytes := UDINT_TO_UINT(#tempValueLength));
	              END_REGION example String
	              
	            ELSIF #columns[#tempColumnLoopCounter].columnName = 'Country' THEN
	              REGION example String
	                //move Bytes to temporary array
	                MOVE_BLK(IN    := #tdsTelegramArray[#statByteAddressCounter],
	                         COUNT := UDINT_TO_UINT(#tempValueLength),
	                         OUT   => #tempByteCharArray[0]);
	                
	                //convert BYTE array to STRING
	                #rows[#tempRowLoopCounter].Country := "LSql_BytesToString"(columnType := #columns[#tempColumnLoopCounter].columnType, byteArray := #tempByteCharArray, numberOfBytes := UDINT_TO_UINT(#tempValueLength));
	              END_REGION example String
	              
	            ELSIF #columns[#tempColumnLoopCounter].columnName = 'CountryCode' THEN
	              REGION example String
	                //move Bytes to temporary array
	                MOVE_BLK(IN    := #tdsTelegramArray[#statByteAddressCounter],
	                         COUNT := UDINT_TO_UINT(#tempValueLength),
	                         OUT   => #tempByteCharArray[0]);
	                
	                //convert BYTE array to STRING
	                #rows[#tempRowLoopCounter].CountryCode := "LSql_BytesToString"(columnType := #columns[#tempColumnLoopCounter].columnType, byteArray := #tempByteCharArray, numberOfBytes := UDINT_TO_UINT(#tempValueLength));
	              END_REGION example String
	              
	            ELSIF #columns[#tempColumnLoopCounter].columnName = 'City' THEN
	              REGION example String
	                //move Bytes to temporary array
	                MOVE_BLK(IN    := #tdsTelegramArray[#statByteAddressCounter],
	                         COUNT := UDINT_TO_UINT(#tempValueLength),
	                         OUT   => #tempByteCharArray[0]);
	                
	                //convert BYTE array to STRING
	                #rows[#tempRowLoopCounter].City := "LSql_BytesToString"(columnType := #columns[#tempColumnLoopCounter].columnType, byteArray := #tempByteCharArray, numberOfBytes := UDINT_TO_UINT(#tempValueLength));
	              END_REGION example String
	              
	            ELSIF #columns[#tempColumnLoopCounter].columnName = 'Taste' THEN
	              REGION example String
	                //move Bytes to temporary array
	                MOVE_BLK(IN    := #tdsTelegramArray[#statByteAddressCounter],
	                         COUNT := UDINT_TO_UINT(#tempValueLength),
	                         OUT   => #tempByteCharArray[0]);
	                
	                //convert BYTE array to STRING
	                #rows[#tempRowLoopCounter].Taste := "LSql_BytesToString"(columnType := #columns[#tempColumnLoopCounter].columnType, byteArray := #tempByteCharArray, numberOfBytes := UDINT_TO_UINT(#tempValueLength));
	              END_REGION example String
	              *)
	              
	            ELSE
	              //column name is not handled by user program case
	              #statWarning := TRUE;
	              
	              //check if there has not been any other major error yet
	              IF (#statStatus = #ERR_NOERROR) THEN
	                #statStatus := #ERR_COULMNS_COLUMNNOTEXISTING;
	              END_IF;
	              
	            END_IF;
	          END_REGION --> use case deserializaition
	          
	          //iterate counter by the column size
	          #statByteAddressCounter += UDINT_TO_DINT(#tempValueLength);
	        END_FOR;
	        
	        //increment counter of deserialized rows
	        #statRowsDeserialized += 1;
	        
	      ELSE
	        //the upper slots of the row array will not be filled with received rows anymore
	        //loop execiution can be ended
	        //the number of valid rows is explicitly given as output parameter
	        //set #statRowsDeserialized to the overall final value so the execution does not go on
	        #statRowsDeserialized := DINT_TO_UDINT(#tempTokenRowsUpperBound - #tempTokenRowsLowerBound + 1);
	        EXIT;
	        
	      END_IF;
	      
	    END_FOR;
	    
	  END_REGION deserialize data
	  
	  //operation completed
	  IF (#statRowsDeserialized >= #tempTokenRowsUpperBound - #tempTokenRowsLowerBound + 1) THEN
	    #statDone := TRUE;
	    #statBusy := FALSE;
	  END_IF;
	  
	ELSIF NOT #execute THEN
	  //no execution, reset static output values
	  #statError := FALSE;
	  #statStatus := #ERR_NOERROR;
	  #statDone := FALSE;
	  #statBusy := FALSE;
	  #statWarning := FALSE;
	  #statRowsDeserialized := 0;
	END_IF;
	
	REGION WRITE OUTPUTS
	END:
	  //finally write static values to outputs
	  #rowOverflow := #statRowOverflow;
	  #status := #statStatus;
	  #error := #statError;
	  #warning := #statWarning;
	  #busy := #statBusy;
	  #done := #statDone;
	END_REGION WRITE OUTPUTS
END_FUNCTION_BLOCK

FUNCTION_BLOCK "Main_Safety_RTG1"   // FB1, F_LAD
{ S7_Optimized_Access := 'TRUE' }
   VAR
      ESTOP1 : ESTOP1;
   END_VAR
BEGIN

REGION Network 1: Estops on electrical cabins
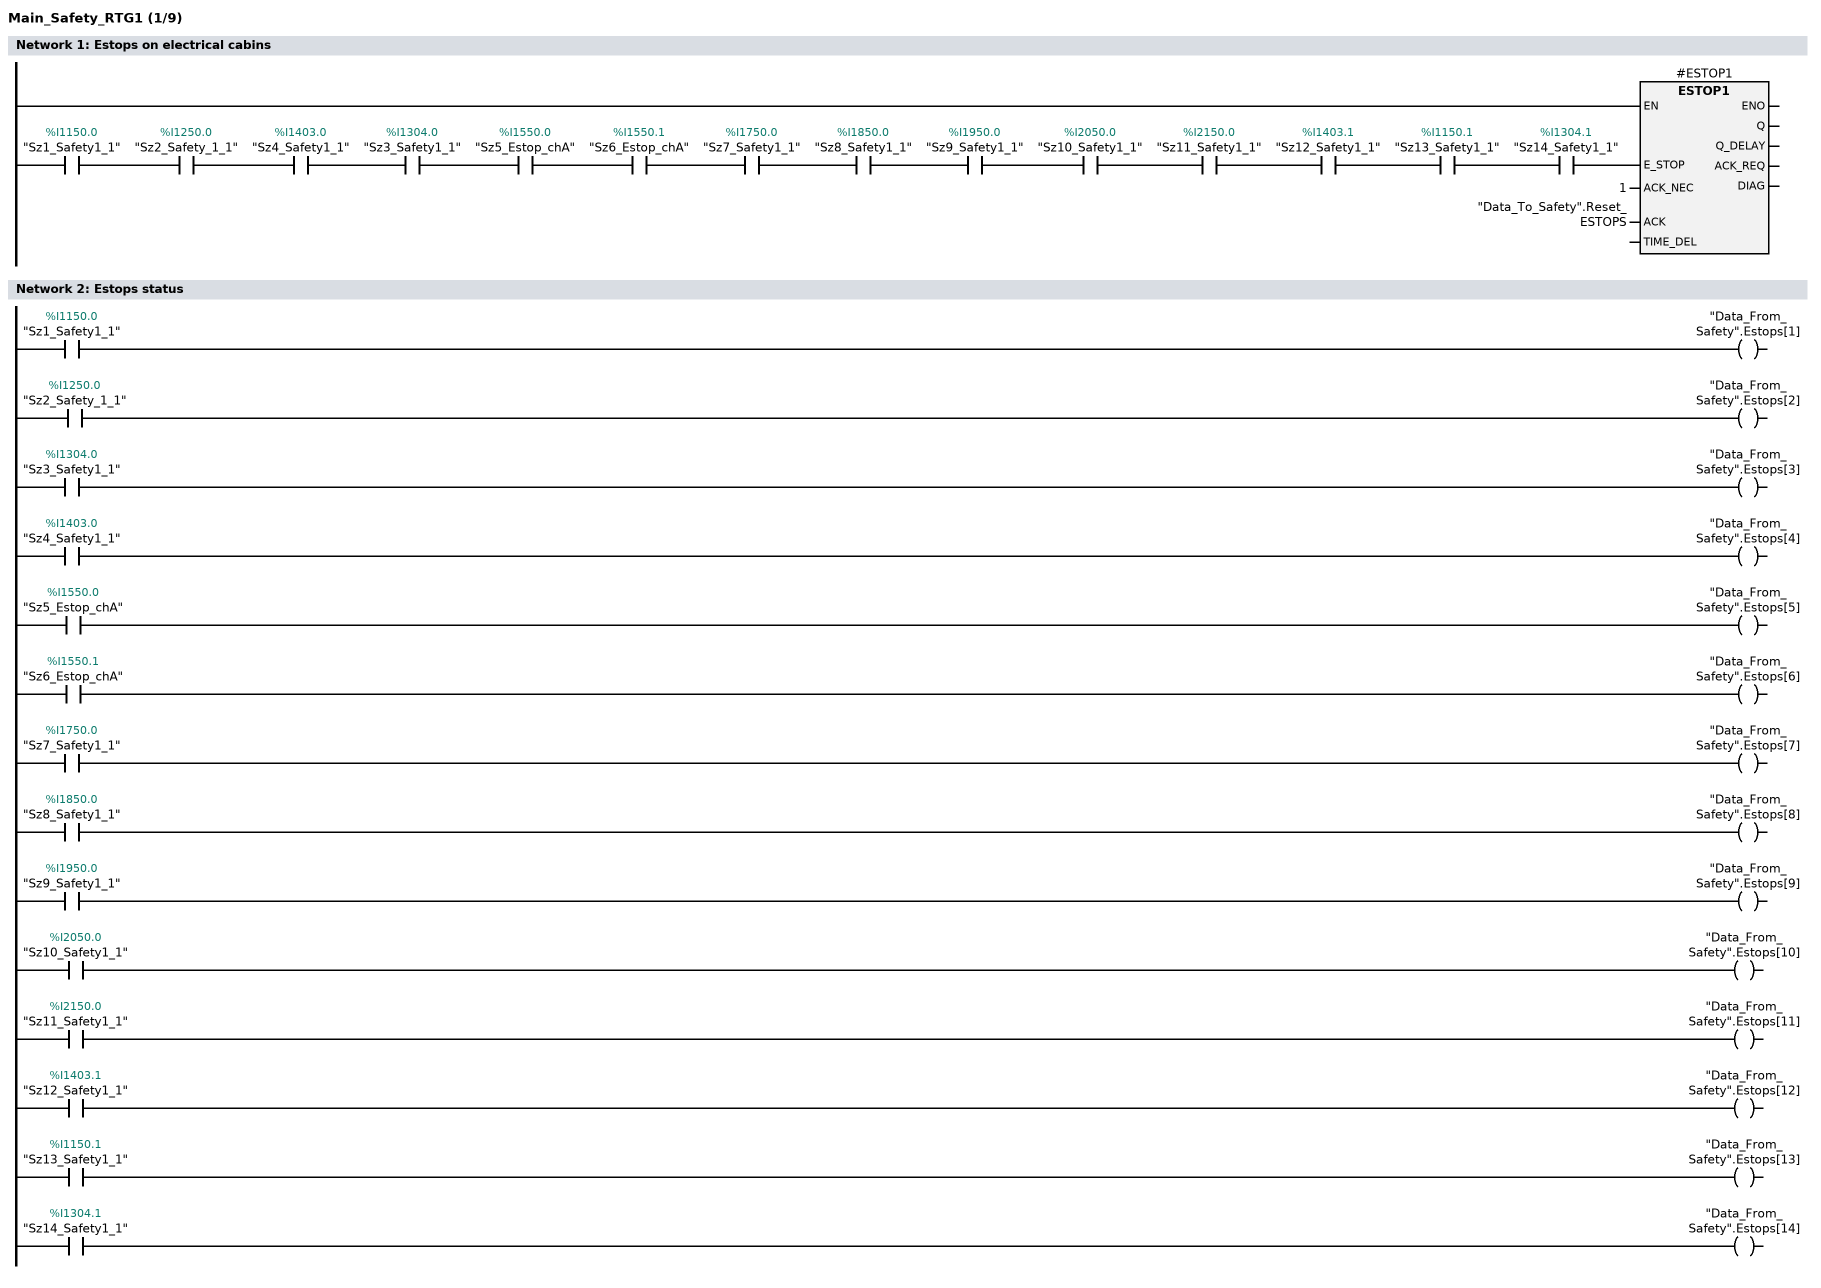
   RUNG wire#powerrail
      #ESTOP1.ESTOP1(E_STOP := wire#w1, ACK_NEC := 1, ACK := "Data_To_Safety".Reset_ESTOPS, TIME_DEL :=, Q =>, Q_DELAY =>, ACK_REQ =>, DIAG =>)
   END_RUNG
   RUNG wire#powerrail
      Contact( "Sz1_Safety1_1" )
      Contact( "Sz2_Safety_1_1" )
      Contact( "Sz4_Safety1_1" )
      Contact( "Sz3_Safety1_1" )
      Contact( "Sz5_Estop_chA" )
      Contact( "Sz6_Estop_chA" )
      Contact( "Sz7_Safety1_1" )
      Contact( "Sz8_Safety1_1" )
      Contact( "Sz9_Safety1_1" )
      Contact( "Sz10_Safety1_1" )
      Contact( "Sz11_Safety1_1" )
      Contact( "Sz12_Safety1_1" )
      Contact( "Sz13_Safety1_1" )
      Contact( "Sz14_Safety1_1" )
   END_RUNG wire#w1
   // the same network as SCL:
   #ESTOP1(E_STOP := "Sz1_Safety1_1" AND "Sz2_Safety_1_1" AND "Sz4_Safety1_1" AND "Sz3_Safety1_1" AND "Sz5_Estop_chA" AND "Sz6_Estop_chA" AND "Sz7_Safety1_1" AND "Sz8_Safety1_1" AND "Sz9_Safety1_1" AND "Sz10_Safety1_1" AND "Sz11_Safety1_1" AND "Sz12_Safety1_1" AND "Sz13_Safety1_1" AND "Sz14_Safety1_1",   // ESTOP1
           ACK_NEC := 1,
           ACK := "Data_To_Safety".Reset_ESTOPS);
END_REGION

REGION Network 2: Estops status
   RUNG wire#powerrail
      Contact( "Sz1_Safety1_1" )
      Coil( "Data_From_Safety".Estops[1] )
   END_RUNG
   RUNG wire#powerrail
      Contact( "Sz2_Safety_1_1" )
      Coil( "Data_From_Safety".Estops[2] )
   END_RUNG
   RUNG wire#powerrail
      Contact( "Sz3_Safety1_1" )
      Coil( "Data_From_Safety".Estops[3] )
   END_RUNG
   RUNG wire#powerrail
      Contact( "Sz4_Safety1_1" )
      Coil( "Data_From_Safety".Estops[4] )
   END_RUNG
   RUNG wire#powerrail
      Contact( "Sz5_Estop_chA" )
      Coil( "Data_From_Safety".Estops[5] )
   END_RUNG
   RUNG wire#powerrail
      Contact( "Sz6_Estop_chA" )
      Coil( "Data_From_Safety".Estops[6] )
   END_RUNG
   RUNG wire#powerrail
      Contact( "Sz7_Safety1_1" )
      Coil( "Data_From_Safety".Estops[7] )
   END_RUNG
   RUNG wire#powerrail
      Contact( "Sz8_Safety1_1" )
      Coil( "Data_From_Safety".Estops[8] )
   END_RUNG
   RUNG wire#powerrail
      Contact( "Sz9_Safety1_1" )
      Coil( "Data_From_Safety".Estops[9] )
   END_RUNG
   RUNG wire#powerrail
      Contact( "Sz10_Safety1_1" )
      Coil( "Data_From_Safety".Estops[10] )
   END_RUNG
   RUNG wire#powerrail
      Contact( "Sz11_Safety1_1" )
      Coil( "Data_From_Safety".Estops[11] )
   END_RUNG
   RUNG wire#powerrail
      Contact( "Sz12_Safety1_1" )
      Coil( "Data_From_Safety".Estops[12] )
   END_RUNG
   RUNG wire#powerrail
      Contact( "Sz13_Safety1_1" )
      Coil( "Data_From_Safety".Estops[13] )
   END_RUNG
   RUNG wire#powerrail
      Contact( "Sz14_Safety1_1" )
      Coil( "Data_From_Safety".Estops[14] )
   END_RUNG
   // the same network as SCL:
   "Data_From_Safety".Estops[1] := "Sz1_Safety1_1";
   "Data_From_Safety".Estops[2] := "Sz2_Safety_1_1";
   "Data_From_Safety".Estops[3] := "Sz3_Safety1_1";
   "Data_From_Safety".Estops[4] := "Sz4_Safety1_1";
   "Data_From_Safety".Estops[5] := "Sz5_Estop_chA";
   "Data_From_Safety".Estops[6] := "Sz6_Estop_chA";
   "Data_From_Safety".Estops[7] := "Sz7_Safety1_1";
   "Data_From_Safety".Estops[8] := "Sz8_Safety1_1";
   "Data_From_Safety".Estops[9] := "Sz9_Safety1_1";
   "Data_From_Safety".Estops[10] := "Sz10_Safety1_1";
   "Data_From_Safety".Estops[11] := "Sz11_Safety1_1";
   "Data_From_Safety".Estops[12] := "Sz12_Safety1_1";
   "Data_From_Safety".Estops[13] := "Sz13_Safety1_1";
   "Data_From_Safety".Estops[14] := "Sz14_Safety1_1";
END_REGION

REGION Network 3: Bumpers SS1_R1
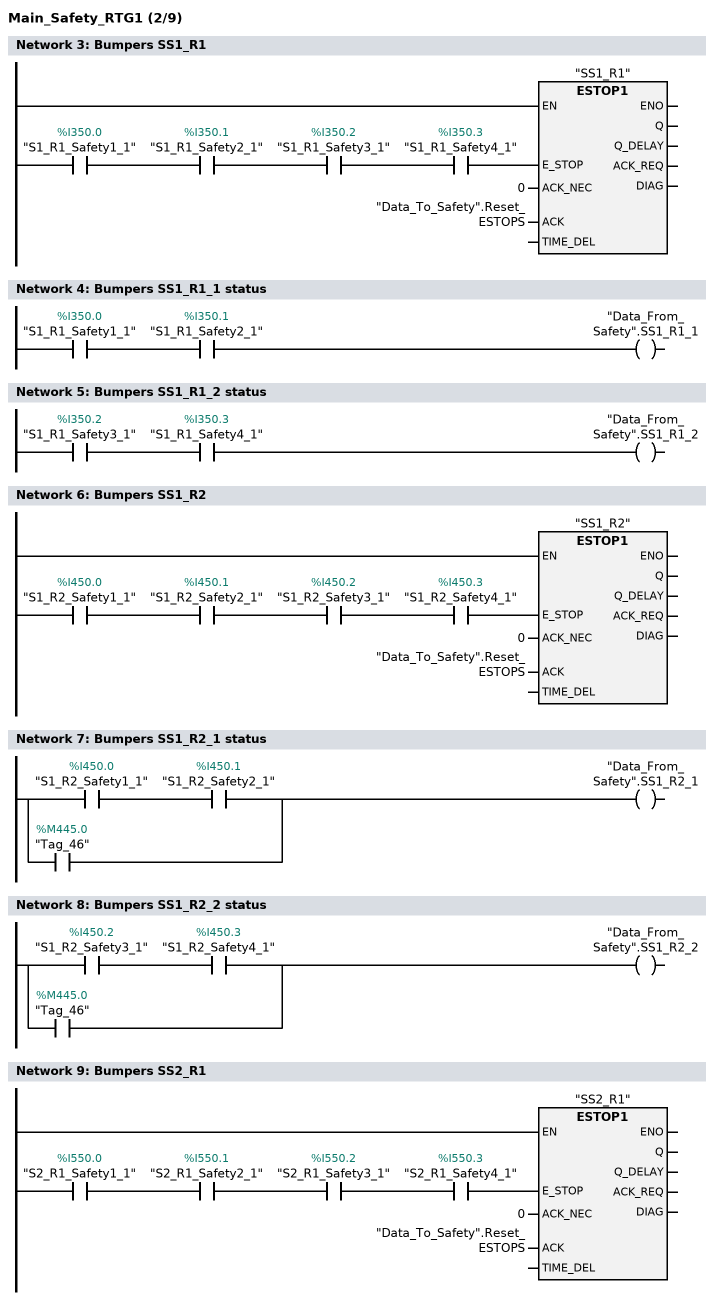
   RUNG wire#powerrail
      "SS1_R1".ESTOP1(E_STOP := wire#w1, ACK_NEC := 0, ACK := "Data_To_Safety".Reset_ESTOPS, TIME_DEL :=, Q =>, Q_DELAY =>, ACK_REQ =>, DIAG =>)
   END_RUNG
   RUNG wire#powerrail
      Contact( "S1_R1_Safety1_1" )
      Contact( "S1_R1_Safety2_1" )
      Contact( "S1_R1_Safety3_1" )
      Contact( "S1_R1_Safety4_1" )
   END_RUNG wire#w1
   // the same network as SCL:
   "SS1_R1"(E_STOP := "S1_R1_Safety1_1" AND "S1_R1_Safety2_1" AND "S1_R1_Safety3_1" AND "S1_R1_Safety4_1",   // ESTOP1
            ACK_NEC := 0,
            ACK := "Data_To_Safety".Reset_ESTOPS);
END_REGION

REGION Network 4: Bumpers SS1_R1_1 status
   RUNG wire#powerrail
      Contact( "S1_R1_Safety1_1" )
      Contact( "S1_R1_Safety2_1" )
      Coil( "Data_From_Safety".SS1_R1_1 )
   END_RUNG
   // the same network as SCL:
   "Data_From_Safety".SS1_R1_1 := "S1_R1_Safety1_1" AND "S1_R1_Safety2_1";
END_REGION

REGION Network 5: Bumpers SS1_R1_2 status
   RUNG wire#powerrail
      Contact( "S1_R1_Safety3_1" )
      Contact( "S1_R1_Safety4_1" )
      Coil( "Data_From_Safety".SS1_R1_2 )
   END_RUNG
   // the same network as SCL:
   "Data_From_Safety".SS1_R1_2 := "S1_R1_Safety3_1" AND "S1_R1_Safety4_1";
END_REGION

REGION Network 6: Bumpers SS1_R2
   RUNG wire#powerrail
      "SS1_R2".ESTOP1(E_STOP := wire#w1, ACK_NEC := 0, ACK := "Data_To_Safety".Reset_ESTOPS, TIME_DEL :=, Q =>, Q_DELAY =>, ACK_REQ =>, DIAG =>)
   END_RUNG
   RUNG wire#powerrail
      Contact( "S1_R2_Safety1_1" )
      Contact( "S1_R2_Safety2_1" )
      Contact( "S1_R2_Safety3_1" )
      Contact( "S1_R2_Safety4_1" )
   END_RUNG wire#w1
   // the same network as SCL:
   "SS1_R2"(E_STOP := "S1_R2_Safety1_1" AND "S1_R2_Safety2_1" AND "S1_R2_Safety3_1" AND "S1_R2_Safety4_1",   // ESTOP1
            ACK_NEC := 0,
            ACK := "Data_To_Safety".Reset_ESTOPS);
END_REGION

REGION Network 7: Bumpers SS1_R2_1 status
   RUNG wire#powerrail
      Contact( "S1_R2_Safety1_1" )
      Contact( "S1_R2_Safety2_1" )
      wire#w1
      Coil( "Data_From_Safety".SS1_R2_1 )
   END_RUNG
   RUNG wire#powerrail
      Contact( "Tag_46" )
   END_RUNG wire#w1
   // the same network as SCL:
   "Data_From_Safety".SS1_R2_1 := ("S1_R2_Safety1_1" AND "S1_R2_Safety2_1") OR "Tag_46";
END_REGION

REGION Network 8: Bumpers SS1_R2_2 status
   RUNG wire#powerrail
      Contact( "S1_R2_Safety3_1" )
      Contact( "S1_R2_Safety4_1" )
      wire#w1
      Coil( "Data_From_Safety".SS1_R2_2 )
   END_RUNG
   RUNG wire#powerrail
      Contact( "Tag_46" )
   END_RUNG wire#w1
   // the same network as SCL:
   "Data_From_Safety".SS1_R2_2 := ("S1_R2_Safety3_1" AND "S1_R2_Safety4_1") OR "Tag_46";
END_REGION

REGION Network 9: Bumpers SS2_R1
   RUNG wire#powerrail
      "SS2_R1".ESTOP1(E_STOP := wire#w1, ACK_NEC := 0, ACK := "Data_To_Safety".Reset_ESTOPS, TIME_DEL :=, Q =>, Q_DELAY =>, ACK_REQ =>, DIAG =>)
   END_RUNG
   RUNG wire#powerrail
      Contact( "S2_R1_Safety1_1" )
      Contact( "S2_R1_Safety2_1" )
      Contact( "S2_R1_Safety3_1" )
      Contact( "S2_R1_Safety4_1" )
   END_RUNG wire#w1
   // the same network as SCL:
   "SS2_R1"(E_STOP := "S2_R1_Safety1_1" AND "S2_R1_Safety2_1" AND "S2_R1_Safety3_1" AND "S2_R1_Safety4_1",   // ESTOP1
            ACK_NEC := 0,
            ACK := "Data_To_Safety".Reset_ESTOPS);
END_REGION

REGION Network 10: Bumpers SS2_R1_1 status
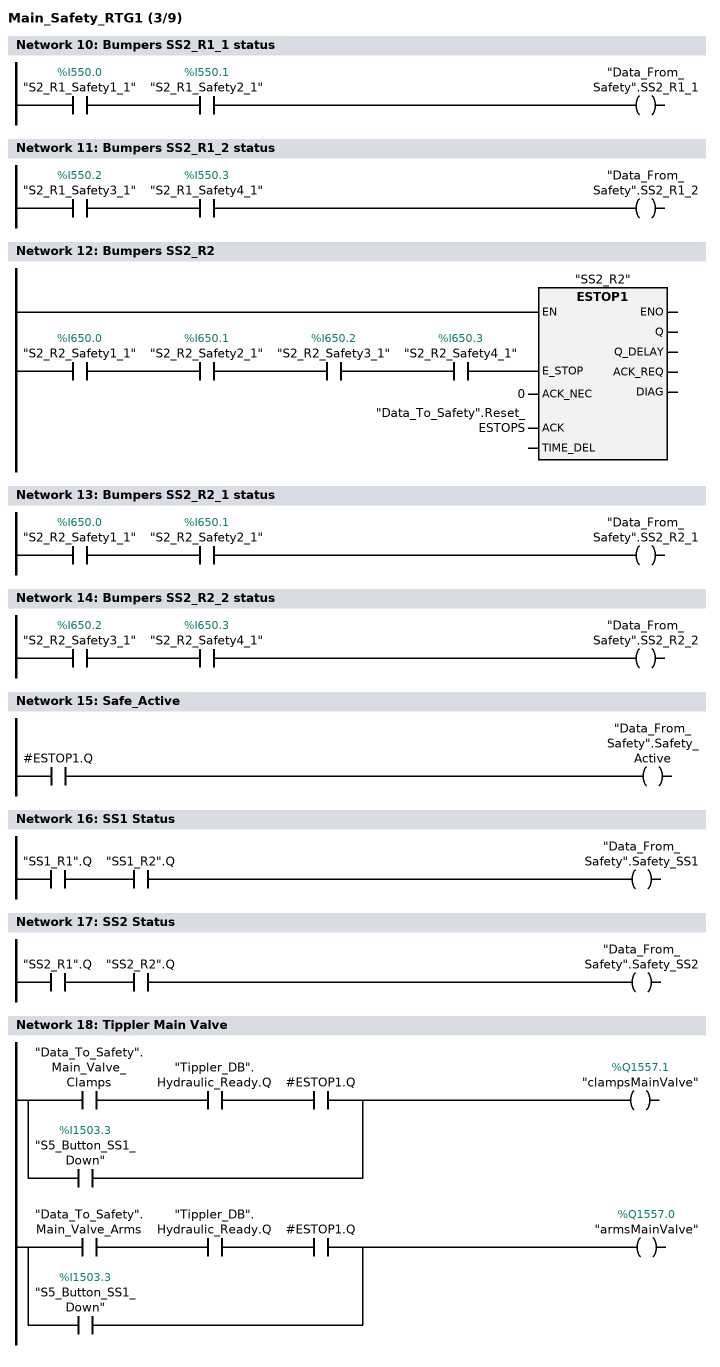
   RUNG wire#powerrail
      Contact( "S2_R1_Safety1_1" )
      Contact( "S2_R1_Safety2_1" )
      Coil( "Data_From_Safety".SS2_R1_1 )
   END_RUNG
   // the same network as SCL:
   "Data_From_Safety".SS2_R1_1 := "S2_R1_Safety1_1" AND "S2_R1_Safety2_1";
END_REGION

REGION Network 11: Bumpers SS2_R1_2 status
   RUNG wire#powerrail
      Contact( "S2_R1_Safety3_1" )
      Contact( "S2_R1_Safety4_1" )
      Coil( "Data_From_Safety".SS2_R1_2 )
   END_RUNG
   // the same network as SCL:
   "Data_From_Safety".SS2_R1_2 := "S2_R1_Safety3_1" AND "S2_R1_Safety4_1";
END_REGION

REGION Network 12: Bumpers SS2_R2
   RUNG wire#powerrail
      "SS2_R2".ESTOP1(E_STOP := wire#w1, ACK_NEC := 0, ACK := "Data_To_Safety".Reset_ESTOPS, TIME_DEL :=, Q =>, Q_DELAY =>, ACK_REQ =>, DIAG =>)
   END_RUNG
   RUNG wire#powerrail
      Contact( "S2_R2_Safety1_1" )
      Contact( "S2_R2_Safety2_1" )
      Contact( "S2_R2_Safety3_1" )
      Contact( "S2_R2_Safety4_1" )
   END_RUNG wire#w1
   // the same network as SCL:
   "SS2_R2"(E_STOP := "S2_R2_Safety1_1" AND "S2_R2_Safety2_1" AND "S2_R2_Safety3_1" AND "S2_R2_Safety4_1",   // ESTOP1
            ACK_NEC := 0,
            ACK := "Data_To_Safety".Reset_ESTOPS);
END_REGION

REGION Network 13: Bumpers SS2_R2_1 status
   RUNG wire#powerrail
      Contact( "S2_R2_Safety1_1" )
      Contact( "S2_R2_Safety2_1" )
      Coil( "Data_From_Safety".SS2_R2_1 )
   END_RUNG
   // the same network as SCL:
   "Data_From_Safety".SS2_R2_1 := "S2_R2_Safety1_1" AND "S2_R2_Safety2_1";
END_REGION

REGION Network 14: Bumpers SS2_R2_2 status
   RUNG wire#powerrail
      Contact( "S2_R2_Safety3_1" )
      Contact( "S2_R2_Safety4_1" )
      Coil( "Data_From_Safety".SS2_R2_2 )
   END_RUNG
   // the same network as SCL:
   "Data_From_Safety".SS2_R2_2 := "S2_R2_Safety3_1" AND "S2_R2_Safety4_1";
END_REGION

REGION Network 15: Safe_Active
   RUNG wire#powerrail
      Contact( #ESTOP1.Q )
      Coil( "Data_From_Safety".Safety_Active )
   END_RUNG
   // the same network as SCL:
   "Data_From_Safety".Safety_Active := #ESTOP1.Q;
END_REGION

REGION Network 16: SS1 Status
   RUNG wire#powerrail
      Contact( "SS1_R1".Q )
      Contact( "SS1_R2".Q )
      Coil( "Data_From_Safety".Safety_SS1 )
   END_RUNG
   // the same network as SCL:
   "Data_From_Safety".Safety_SS1 := "SS1_R1".Q AND "SS1_R2".Q;
END_REGION

REGION Network 17: SS2 Status
   RUNG wire#powerrail
      Contact( "SS2_R1".Q )
      Contact( "SS2_R2".Q )
      Coil( "Data_From_Safety".Safety_SS2 )
   END_RUNG
   // the same network as SCL:
   "Data_From_Safety".Safety_SS2 := "SS2_R1".Q AND "SS2_R2".Q;
END_REGION

REGION Network 18: Tippler Main Valve
   RUNG wire#powerrail
      Contact( "Data_To_Safety".Main_Valve_Clamps )
      Contact( "Tippler_DB".Hydraulic_Ready.Q )
      Contact( #ESTOP1.Q )
      wire#w1
      Coil( "clampsMainValve" )
   END_RUNG
   RUNG wire#powerrail
      Contact( "S5_Button_SS1_Down" )
   END_RUNG wire#w1
   RUNG wire#powerrail
      Contact( "Data_To_Safety".Main_Valve_Arms )
      Contact( "Tippler_DB".Hydraulic_Ready.Q )
      Contact( #ESTOP1.Q )
      wire#w2
      Coil( "armsMainValve" )
   END_RUNG
   RUNG wire#powerrail
      Contact( "S5_Button_SS1_Down" )
   END_RUNG wire#w2
   // the same network as SCL:
   "clampsMainValve" := ("Data_To_Safety".Main_Valve_Clamps AND "Tippler_DB".Hydraulic_Ready.Q AND #ESTOP1.Q) OR "S5_Button_SS1_Down";
   "armsMainValve" := ("Data_To_Safety".Main_Valve_Arms AND "Tippler_DB".Hydraulic_Ready.Q AND #ESTOP1.Q) OR "S5_Button_SS1_Down";
END_REGION

REGION Network 19: S0_R1, S0_R2
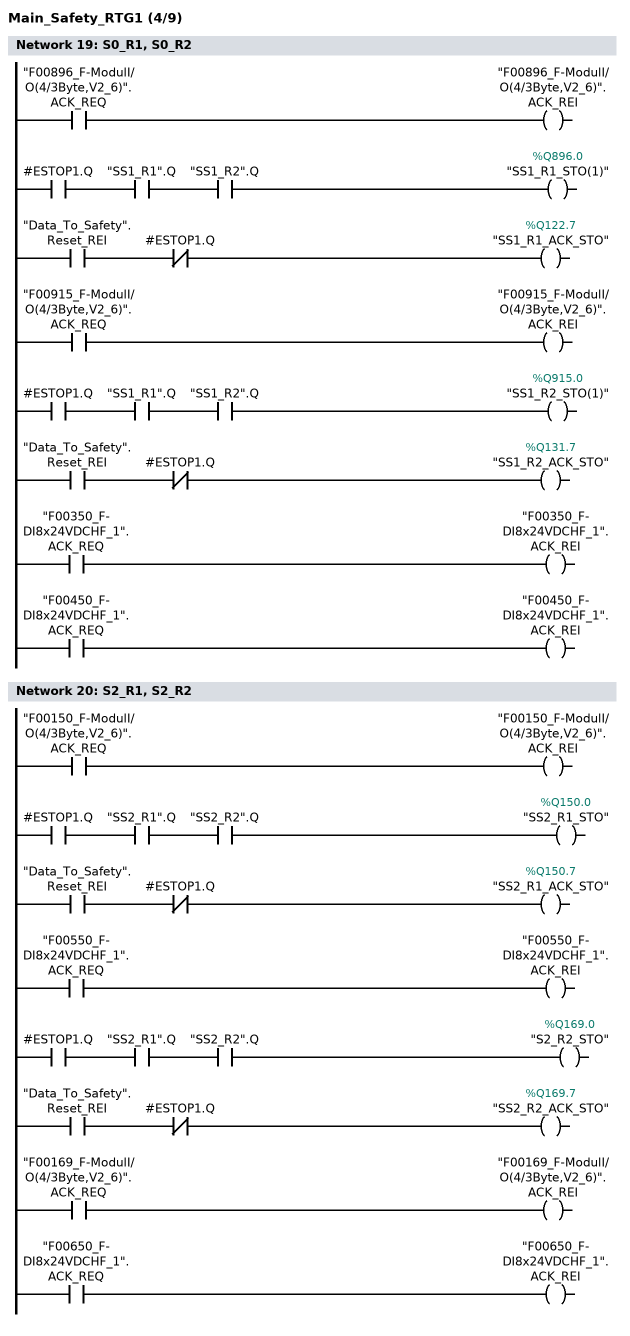
   RUNG wire#powerrail
      Contact( "F00896_F-ModulI/O(4/3Byte,V2_6)".ACK_REQ )
      Coil( "F00896_F-ModulI/O(4/3Byte,V2_6)".ACK_REI )
   END_RUNG
   RUNG wire#powerrail
      Contact( #ESTOP1.Q )
      Contact( "SS1_R1".Q )
      Contact( "SS1_R2".Q )
      Coil( "SS1_R1_STO(1)" )
   END_RUNG
   RUNG wire#powerrail
      Contact( "Data_To_Safety".Reset_REI )
      I_Contact( #ESTOP1.Q )
      Coil( "SS1_R1_ACK_STO" )
   END_RUNG
   RUNG wire#powerrail
      Contact( "F00915_F-ModulI/O(4/3Byte,V2_6)".ACK_REQ )
      Coil( "F00915_F-ModulI/O(4/3Byte,V2_6)".ACK_REI )
   END_RUNG
   RUNG wire#powerrail
      Contact( #ESTOP1.Q )
      Contact( "SS1_R1".Q )
      Contact( "SS1_R2".Q )
      Coil( "SS1_R2_STO(1)" )
   END_RUNG
   RUNG wire#powerrail
      Contact( "Data_To_Safety".Reset_REI )
      I_Contact( #ESTOP1.Q )
      Coil( "SS1_R2_ACK_STO" )
   END_RUNG
   RUNG wire#powerrail
      Contact( "F00350_F-DI8x24VDCHF_1".ACK_REQ )
      Coil( "F00350_F-DI8x24VDCHF_1".ACK_REI )
   END_RUNG
   RUNG wire#powerrail
      Contact( "F00450_F-DI8x24VDCHF_1".ACK_REQ )
      Coil( "F00450_F-DI8x24VDCHF_1".ACK_REI )
   END_RUNG
   // the same network as SCL:
   "F00896_F-ModulI/O(4/3Byte,V2_6)".ACK_REI := "F00896_F-ModulI/O(4/3Byte,V2_6)".ACK_REQ;
   "SS1_R1_STO(1)" := #ESTOP1.Q AND "SS1_R1".Q AND "SS1_R2".Q;
   "SS1_R1_ACK_STO" := "Data_To_Safety".Reset_REI AND NOT #ESTOP1.Q;
   "F00915_F-ModulI/O(4/3Byte,V2_6)".ACK_REI := "F00915_F-ModulI/O(4/3Byte,V2_6)".ACK_REQ;
   "SS1_R2_STO(1)" := #ESTOP1.Q AND "SS1_R1".Q AND "SS1_R2".Q;
   "SS1_R2_ACK_STO" := "Data_To_Safety".Reset_REI AND NOT #ESTOP1.Q;
   "F00350_F-DI8x24VDCHF_1".ACK_REI := "F00350_F-DI8x24VDCHF_1".ACK_REQ;
   "F00450_F-DI8x24VDCHF_1".ACK_REI := "F00450_F-DI8x24VDCHF_1".ACK_REQ;
END_REGION

REGION Network 20: S2_R1, S2_R2
   RUNG wire#powerrail
      Contact( "F00150_F-ModulI/O(4/3Byte,V2_6)".ACK_REQ )
      Coil( "F00150_F-ModulI/O(4/3Byte,V2_6)".ACK_REI )
   END_RUNG
   RUNG wire#powerrail
      Contact( #ESTOP1.Q )
      Contact( "SS2_R1".Q )
      Contact( "SS2_R2".Q )
      Coil( "SS2_R1_STO" )
   END_RUNG
   RUNG wire#powerrail
      Contact( "Data_To_Safety".Reset_REI )
      I_Contact( #ESTOP1.Q )
      Coil( "SS2_R1_ACK_STO" )
   END_RUNG
   RUNG wire#powerrail
      Contact( "F00550_F-DI8x24VDCHF_1".ACK_REQ )
      Coil( "F00550_F-DI8x24VDCHF_1".ACK_REI )
   END_RUNG
   RUNG wire#powerrail
      Contact( #ESTOP1.Q )
      Contact( "SS2_R1".Q )
      Contact( "SS2_R2".Q )
      Coil( "S2_R2_STO" )
   END_RUNG
   RUNG wire#powerrail
      Contact( "Data_To_Safety".Reset_REI )
      I_Contact( #ESTOP1.Q )
      Coil( "SS2_R2_ACK_STO" )
   END_RUNG
   RUNG wire#powerrail
      Contact( "F00169_F-ModulI/O(4/3Byte,V2_6)".ACK_REQ )
      Coil( "F00169_F-ModulI/O(4/3Byte,V2_6)".ACK_REI )
   END_RUNG
   RUNG wire#powerrail
      Contact( "F00650_F-DI8x24VDCHF_1".ACK_REQ )
      Coil( "F00650_F-DI8x24VDCHF_1".ACK_REI )
   END_RUNG
   // the same network as SCL:
   "F00150_F-ModulI/O(4/3Byte,V2_6)".ACK_REI := "F00150_F-ModulI/O(4/3Byte,V2_6)".ACK_REQ;
   "SS2_R1_STO" := #ESTOP1.Q AND "SS2_R1".Q AND "SS2_R2".Q;
   "SS2_R1_ACK_STO" := "Data_To_Safety".Reset_REI AND NOT #ESTOP1.Q;
   "F00550_F-DI8x24VDCHF_1".ACK_REI := "F00550_F-DI8x24VDCHF_1".ACK_REQ;
   "S2_R2_STO" := #ESTOP1.Q AND "SS2_R1".Q AND "SS2_R2".Q;
   "SS2_R2_ACK_STO" := "Data_To_Safety".Reset_REI AND NOT #ESTOP1.Q;
   "F00169_F-ModulI/O(4/3Byte,V2_6)".ACK_REI := "F00169_F-ModulI/O(4/3Byte,V2_6)".ACK_REQ;
   "F00650_F-DI8x24VDCHF_1".ACK_REI := "F00650_F-DI8x24VDCHF_1".ACK_REQ;
END_REGION

REGION Network 21: 1=Acknowledgment for reintegration
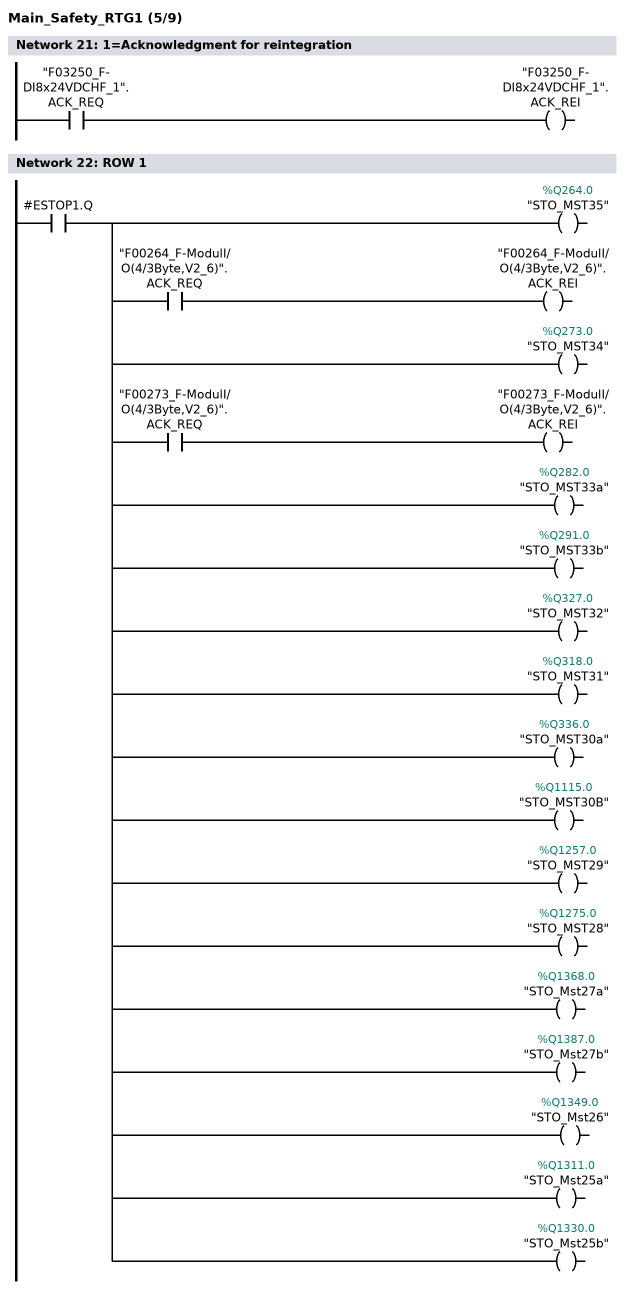
   RUNG wire#powerrail
      Contact( "F03250_F-DI8x24VDCHF_1".ACK_REQ )
      Coil( "F03250_F-DI8x24VDCHF_1".ACK_REI )
   END_RUNG
   // the same network as SCL:
   "F03250_F-DI8x24VDCHF_1".ACK_REI := "F03250_F-DI8x24VDCHF_1".ACK_REQ;
END_REGION

REGION Network 22: ROW 1
   RUNG wire#powerrail
      Contact( #ESTOP1.Q )
      wire#w1
      Coil( "STO_MST35" )
   END_RUNG
   RUNG wire#w1
      Contact( "F00264_F-ModulI/O(4/3Byte,V2_6)".ACK_REQ )
      Coil( "F00264_F-ModulI/O(4/3Byte,V2_6)".ACK_REI )
   END_RUNG
   RUNG wire#w1
      Coil( "STO_MST34" )
   END_RUNG
   RUNG wire#w1
      Contact( "F00273_F-ModulI/O(4/3Byte,V2_6)".ACK_REQ )
      Coil( "F00273_F-ModulI/O(4/3Byte,V2_6)".ACK_REI )
   END_RUNG
   RUNG wire#w1
      Coil( "STO_MST33a" )
   END_RUNG
   RUNG wire#w1
      Coil( "STO_MST33b" )
   END_RUNG
   RUNG wire#w1
      Coil( "STO_MST32" )
   END_RUNG
   RUNG wire#w1
      Coil( "STO_MST31" )
   END_RUNG
   RUNG wire#w1
      Coil( "STO_MST30a" )
   END_RUNG
   RUNG wire#w1
      Coil( "STO_MST30B" )
   END_RUNG
   RUNG wire#w1
      Coil( "STO_MST29" )
   END_RUNG
   RUNG wire#w1
      Coil( "STO_MST28" )
   END_RUNG
   RUNG wire#w1
      Coil( "STO_Mst27a" )
   END_RUNG
   RUNG wire#w1
      Coil( "STO_Mst27b" )
   END_RUNG
   RUNG wire#w1
      Coil( "STO_Mst26" )
   END_RUNG
   RUNG wire#w1
      Coil( "STO_Mst25a" )
   END_RUNG
   RUNG wire#w1
      Coil( "STO_Mst25b" )
   END_RUNG
   // the same network as SCL:
   "STO_MST35" := #ESTOP1.Q;
   "F00264_F-ModulI/O(4/3Byte,V2_6)".ACK_REI := #ESTOP1.Q AND "F00264_F-ModulI/O(4/3Byte,V2_6)".ACK_REQ;
   "STO_MST34" := #ESTOP1.Q;
   "F00273_F-ModulI/O(4/3Byte,V2_6)".ACK_REI := #ESTOP1.Q AND "F00273_F-ModulI/O(4/3Byte,V2_6)".ACK_REQ;
   "STO_MST33a" := #ESTOP1.Q;
   "STO_MST33b" := #ESTOP1.Q;
   "STO_MST32" := #ESTOP1.Q;
   "STO_MST31" := #ESTOP1.Q;
   "STO_MST30a" := #ESTOP1.Q;
   "STO_MST30B" := #ESTOP1.Q;
   "STO_MST29" := #ESTOP1.Q;
   "STO_MST28" := #ESTOP1.Q;
   "STO_Mst27a" := #ESTOP1.Q;
   "STO_Mst27b" := #ESTOP1.Q;
   "STO_Mst26" := #ESTOP1.Q;
   "STO_Mst25a" := #ESTOP1.Q;
   "STO_Mst25b" := #ESTOP1.Q;
END_REGION

REGION Network 23: ROW 2
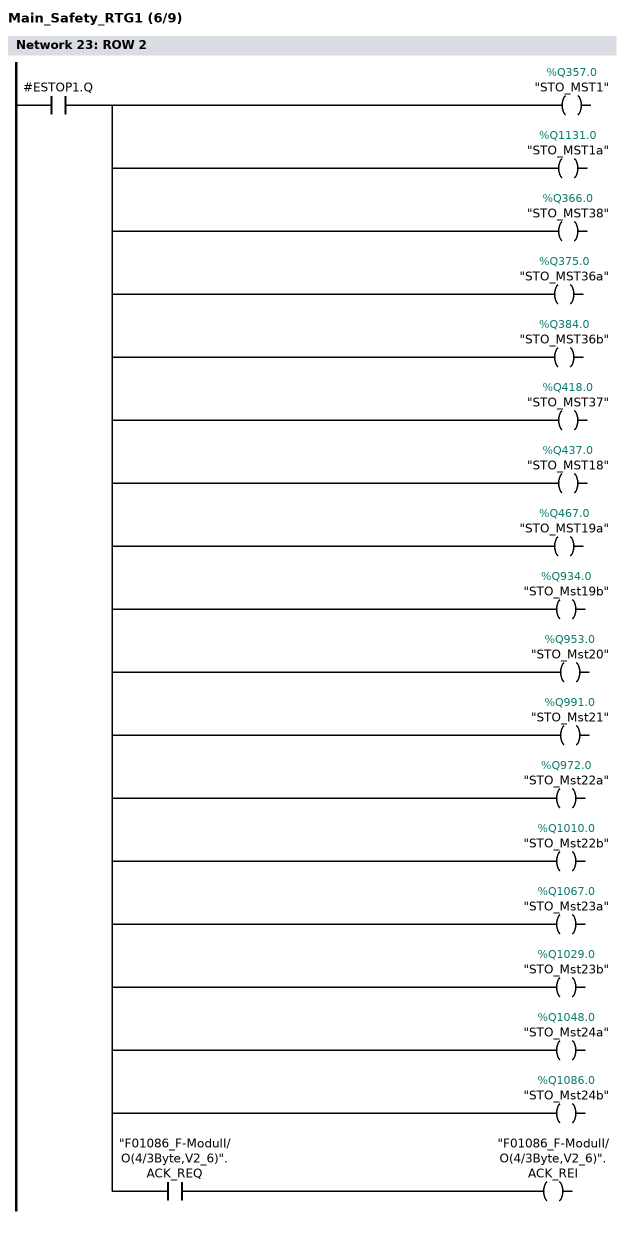
   RUNG wire#powerrail
      Contact( #ESTOP1.Q )
      wire#w1
      Coil( "STO_MST1" )
   END_RUNG
   RUNG wire#w1
      Coil( "STO_MST1a" )
   END_RUNG
   RUNG wire#w1
      Coil( "STO_MST38" )
   END_RUNG
   RUNG wire#w1
      Coil( "STO_MST36a" )
   END_RUNG
   RUNG wire#w1
      Coil( "STO_MST36b" )
   END_RUNG
   RUNG wire#w1
      Coil( "STO_MST37" )
   END_RUNG
   RUNG wire#w1
      Coil( "STO_MST18" )
   END_RUNG
   RUNG wire#w1
      Coil( "STO_MST19a" )
   END_RUNG
   RUNG wire#w1
      Coil( "STO_Mst19b" )
   END_RUNG
   RUNG wire#w1
      Coil( "STO_Mst20" )
   END_RUNG
   RUNG wire#w1
      Coil( "STO_Mst21" )
   END_RUNG
   RUNG wire#w1
      Coil( "STO_Mst22a" )
   END_RUNG
   RUNG wire#w1
      Coil( "STO_Mst22b" )
   END_RUNG
   RUNG wire#w1
      Coil( "STO_Mst23a" )
   END_RUNG
   RUNG wire#w1
      Coil( "STO_Mst23b" )
   END_RUNG
   RUNG wire#w1
      Coil( "STO_Mst24a" )
   END_RUNG
   RUNG wire#w1
      Coil( "STO_Mst24b" )
   END_RUNG
   RUNG wire#w1
      Contact( "F01086_F-ModulI/O(4/3Byte,V2_6)".ACK_REQ )
      Coil( "F01086_F-ModulI/O(4/3Byte,V2_6)".ACK_REI )
   END_RUNG
   // the same network as SCL:
   "STO_MST1" := #ESTOP1.Q;
   "STO_MST1a" := #ESTOP1.Q;
   "STO_MST38" := #ESTOP1.Q;
   "STO_MST36a" := #ESTOP1.Q;
   "STO_MST36b" := #ESTOP1.Q;
   "STO_MST37" := #ESTOP1.Q;
   "STO_MST18" := #ESTOP1.Q;
   "STO_MST19a" := #ESTOP1.Q;
   "STO_Mst19b" := #ESTOP1.Q;
   "STO_Mst20" := #ESTOP1.Q;
   "STO_Mst21" := #ESTOP1.Q;
   "STO_Mst22a" := #ESTOP1.Q;
   "STO_Mst22b" := #ESTOP1.Q;
   "STO_Mst23a" := #ESTOP1.Q;
   "STO_Mst23b" := #ESTOP1.Q;
   "STO_Mst24a" := #ESTOP1.Q;
   "STO_Mst24b" := #ESTOP1.Q;
   "F01086_F-ModulI/O(4/3Byte,V2_6)".ACK_REI := #ESTOP1.Q AND "F01086_F-ModulI/O(4/3Byte,V2_6)".ACK_REQ;
END_REGION

REGION Network 24: ROW 4
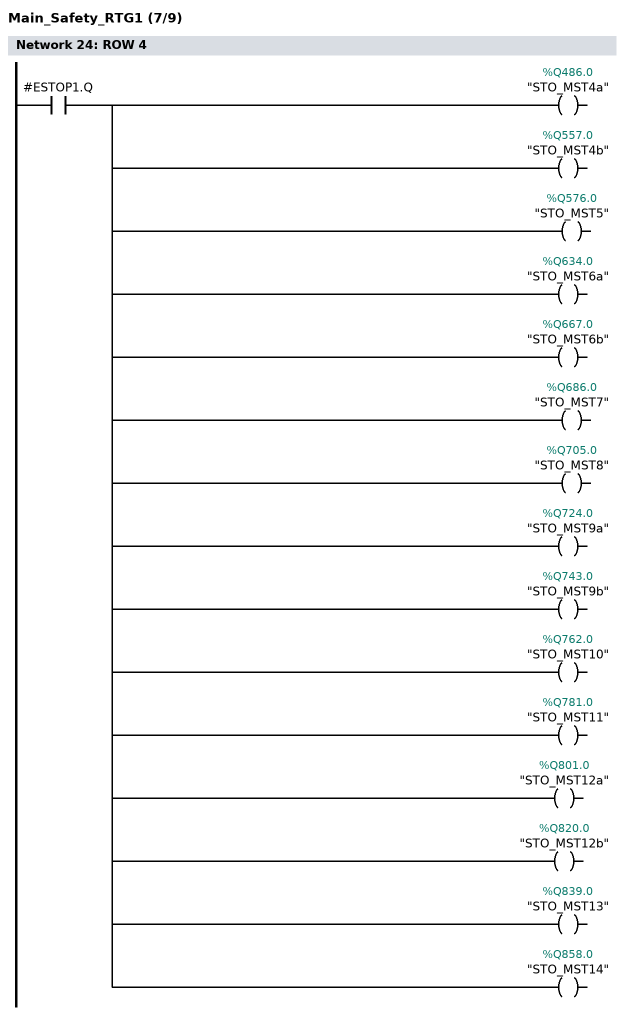
   RUNG wire#powerrail
      Contact( #ESTOP1.Q )
      wire#w1
      Coil( "STO_MST4a" )
   END_RUNG
   RUNG wire#w1
      Coil( "STO_MST4b" )
   END_RUNG
   RUNG wire#w1
      Coil( "STO_MST5" )
   END_RUNG
   RUNG wire#w1
      Coil( "STO_MST6a" )
   END_RUNG
   RUNG wire#w1
      Coil( "STO_MST6b" )
   END_RUNG
   RUNG wire#w1
      Coil( "STO_MST7" )
   END_RUNG
   RUNG wire#w1
      Coil( "STO_MST8" )
   END_RUNG
   RUNG wire#w1
      Coil( "STO_MST9a" )
   END_RUNG
   RUNG wire#w1
      Coil( "STO_MST9b" )
   END_RUNG
   RUNG wire#w1
      Coil( "STO_MST10" )
   END_RUNG
   RUNG wire#w1
      Coil( "STO_MST11" )
   END_RUNG
   RUNG wire#w1
      Coil( "STO_MST12a" )
   END_RUNG
   RUNG wire#w1
      Coil( "STO_MST12b" )
   END_RUNG
   RUNG wire#w1
      Coil( "STO_MST13" )
   END_RUNG
   RUNG wire#w1
      Coil( "STO_MST14" )
   END_RUNG
   // the same network as SCL:
   "STO_MST4a" := #ESTOP1.Q;
   "STO_MST4b" := #ESTOP1.Q;
   "STO_MST5" := #ESTOP1.Q;
   "STO_MST6a" := #ESTOP1.Q;
   "STO_MST6b" := #ESTOP1.Q;
   "STO_MST7" := #ESTOP1.Q;
   "STO_MST8" := #ESTOP1.Q;
   "STO_MST9a" := #ESTOP1.Q;
   "STO_MST9b" := #ESTOP1.Q;
   "STO_MST10" := #ESTOP1.Q;
   "STO_MST11" := #ESTOP1.Q;
   "STO_MST12a" := #ESTOP1.Q;
   "STO_MST12b" := #ESTOP1.Q;
   "STO_MST13" := #ESTOP1.Q;
   "STO_MST14" := #ESTOP1.Q;
END_REGION

REGION Network 25: CS
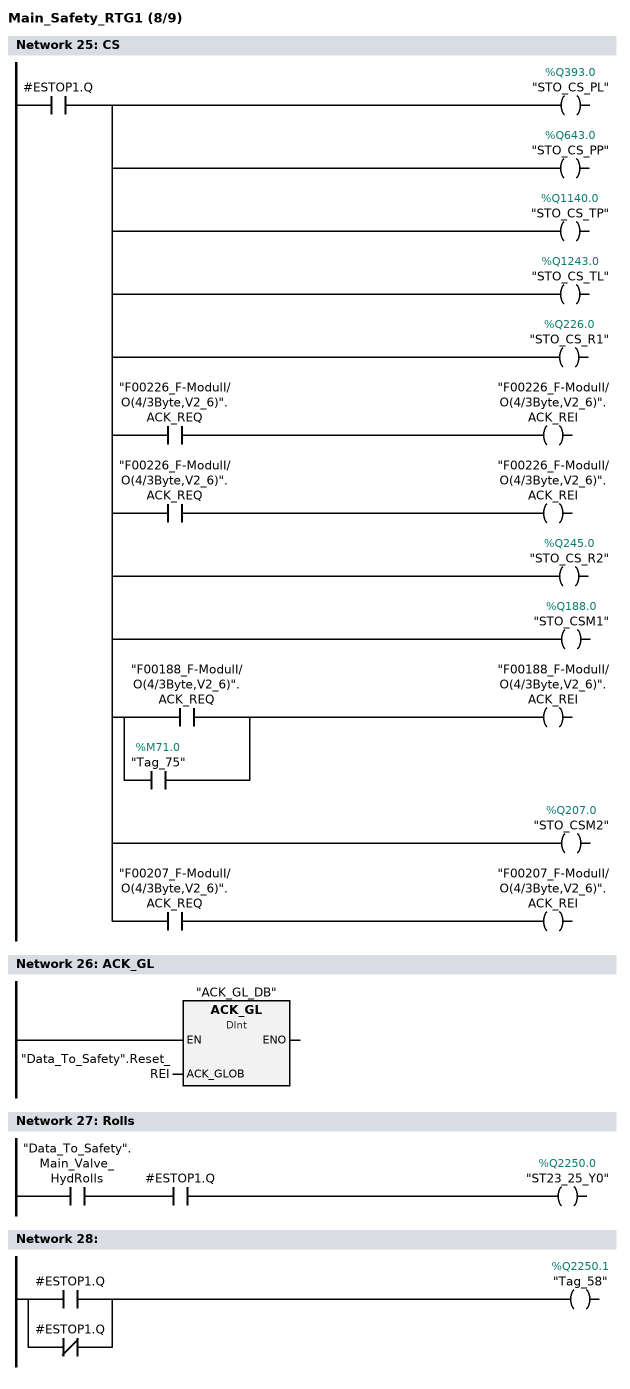
   RUNG wire#powerrail
      Contact( #ESTOP1.Q )
      wire#w1
      Coil( "STO_CS_PL" )
   END_RUNG
   RUNG wire#w1
      Coil( "STO_CS_PP" )
   END_RUNG
   RUNG wire#w1
      Coil( "STO_CS_TP" )
   END_RUNG
   RUNG wire#w1
      Coil( "STO_CS_TL" )
   END_RUNG
   RUNG wire#w1
      Coil( "STO_CS_R1" )
   END_RUNG
   RUNG wire#w1
      Contact( "F00226_F-ModulI/O(4/3Byte,V2_6)".ACK_REQ )
      Coil( "F00226_F-ModulI/O(4/3Byte,V2_6)".ACK_REI )
   END_RUNG
   RUNG wire#w1
      Contact( "F00226_F-ModulI/O(4/3Byte,V2_6)".ACK_REQ )
      Coil( "F00226_F-ModulI/O(4/3Byte,V2_6)".ACK_REI )
   END_RUNG
   RUNG wire#w1
      Coil( "STO_CS_R2" )
   END_RUNG
   RUNG wire#w1
      Coil( "STO_CSM1" )
   END_RUNG
   RUNG wire#w1
      Contact( "F00188_F-ModulI/O(4/3Byte,V2_6)".ACK_REQ )
      wire#w2
      Coil( "F00188_F-ModulI/O(4/3Byte,V2_6)".ACK_REI )
   END_RUNG
   RUNG wire#w1
      Contact( "Tag_75" )
   END_RUNG wire#w2
   RUNG wire#w1
      Coil( "STO_CSM2" )
   END_RUNG
   RUNG wire#w1
      Contact( "F00207_F-ModulI/O(4/3Byte,V2_6)".ACK_REQ )
      Coil( "F00207_F-ModulI/O(4/3Byte,V2_6)".ACK_REI )
   END_RUNG
   // the same network as SCL:
   "STO_CS_PL" := #ESTOP1.Q;
   "STO_CS_PP" := #ESTOP1.Q;
   "STO_CS_TP" := #ESTOP1.Q;
   "STO_CS_TL" := #ESTOP1.Q;
   "STO_CS_R1" := #ESTOP1.Q;
   "F00226_F-ModulI/O(4/3Byte,V2_6)".ACK_REI := #ESTOP1.Q AND "F00226_F-ModulI/O(4/3Byte,V2_6)".ACK_REQ;
   "F00226_F-ModulI/O(4/3Byte,V2_6)".ACK_REI := #ESTOP1.Q AND "F00226_F-ModulI/O(4/3Byte,V2_6)".ACK_REQ;
   "STO_CS_R2" := #ESTOP1.Q;
   "STO_CSM1" := #ESTOP1.Q;
   "F00188_F-ModulI/O(4/3Byte,V2_6)".ACK_REI := #ESTOP1.Q AND ("F00188_F-ModulI/O(4/3Byte,V2_6)".ACK_REQ OR "Tag_75");
   "STO_CSM2" := #ESTOP1.Q;
   "F00207_F-ModulI/O(4/3Byte,V2_6)".ACK_REI := #ESTOP1.Q AND "F00207_F-ModulI/O(4/3Byte,V2_6)".ACK_REQ;
END_REGION

REGION Network 26: ACK_GL
   RUNG wire#powerrail
      { S7_Templates := "codedbool_type := DInt" } "ACK_GL_DB".ACK_GL(ACK_GLOB := "Data_To_Safety".Reset_REI)
   END_RUNG
   // the same network as SCL:
   "ACK_GL_DB"(ACK_GLOB := "Data_To_Safety".Reset_REI);   // ACK_GL
END_REGION

REGION Network 27: Rolls
   RUNG wire#powerrail
      Contact( "Data_To_Safety".Main_Valve_HydRolls )
      Contact( #ESTOP1.Q )
      Coil( "ST23_25_Y0" )
   END_RUNG
   // the same network as SCL:
   "ST23_25_Y0" := "Data_To_Safety".Main_Valve_HydRolls AND #ESTOP1.Q;
END_REGION

REGION Network 28
   RUNG wire#powerrail
      Contact( #ESTOP1.Q )
      wire#w1
      Coil( "Tag_58" )
   END_RUNG
   RUNG wire#powerrail
      I_Contact( #ESTOP1.Q )
   END_RUNG wire#w1
   // the same network as SCL:
   "Tag_58" := #ESTOP1.Q OR NOT #ESTOP1.Q;
END_REGION

REGION Network 29: 1=Acknowledgment for reintegration
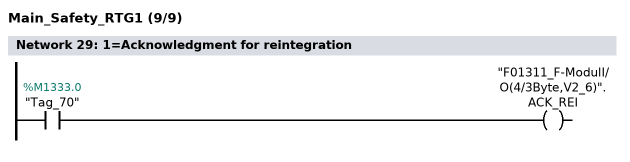
   RUNG wire#powerrail
      Contact( "Tag_70" )
      Coil( "F01311_F-ModulI/O(4/3Byte,V2_6)".ACK_REI )
   END_RUNG
   // the same network as SCL:
   "F01311_F-ModulI/O(4/3Byte,V2_6)".ACK_REI := "Tag_70";
END_REGION
END_FUNCTION_BLOCK

FUNCTION_BLOCK "CentralShifter_HMI_Move_Pallet"
{ S7_Optimized_Access := 'TRUE' }
VERSION : 0.1
   VAR 
      Column_Start : SInt;
      Column_Destination : SInt;
      Row_Start : SInt;
      Row_Destination : SInt;
      Step : SInt;
   END_VAR


BEGIN
END_FUNCTION_BLOCK

FUNCTION "Clean_Movment" : Void
{ S7_Optimized_Access := 'TRUE' }
VERSION : 0.1
   VAR_IN_OUT 
      Arr : Array[1..12] of Bool;
   END_VAR

   VAR_TEMP 
      i : SInt;
      Found : Bool;
   END_VAR


BEGIN
	FOR #i := 1 TO 12 DO
	    IF #Arr[#i] AND NOT #Found THEN
	        #Found := TRUE;   // pierwszy TRUE zostaje
	    ELSE
	        #Arr[#i] := FALSE; // reszta reset
	    END_IF;
	END_FOR;
END_FUNCTION

DATA_BLOCK "CentralShifter_DB"   // DB31
// stored: InstanceOfName CentralShifter, InstanceOfType FB
"CentralShifter"
BEGIN
   CentralShifter_SideShifters_Instance.Stations[12].RL_H3_Pos := 13515;
   CentralShifter_SideShifters_Instance.Stations[13].RL_H3_Pos := 13500;
   CentralShifter_SideShifters_Instance.Stations[12..13].RR_H3_Pos := 13525;
   CentralShifter_SideShifters_Instance.Stations[12].RL_Mid_Pos := 7932;
   CentralShifter_SideShifters_Instance.Stations[13].RL_Mid_Pos := 7916;
   CentralShifter_SideShifters_Instance.Stations[12].RR_Mid_Pos := 7932;
   CentralShifter_SideShifters_Instance.Stations[13].RR_Mid_Pos := 7939;
   CentralShifter_SideShifters_Instance.Stations[12].RL_H5_Pos := 1924;
   CentralShifter_SideShifters_Instance.Stations[13].RL_H5_Pos := 1918;
   CentralShifter_SideShifters_Instance.Stations[12].RR_H5_Pos := 1934;
   CentralShifter_SideShifters_Instance.Stations[13].RR_H5_Pos := 1915;
   CentralShifter_SideShifters_Instance.Stations[12].Correction := 10;
   CentralShifter_SideShifters_Instance.Stations[13].Correction := 15;
END_DATA_BLOCK

DATA_BLOCK "SimpleEnc_DB"   // DB39
// stored: InstanceOfName SimpleEnc, InstanceOfType FB
"SimpleEnc"
BEGIN
END_DATA_BLOCK

DATA_BLOCK "TorqueFB_TEL750_DB"   // DB45
// stored: InstanceOfName TorqueFB_TEL750, InstanceOfType FB
"TorqueFB_TEL750"
BEGIN
END_DATA_BLOCK

DATA_BLOCK "DB_CC_Main"   // DB101
// stored: AutoNumber false, InstanceOfName CC_Main, InstanceOfType FB
"CC_Main"
BEGIN
END_DATA_BLOCK

DATA_BLOCK "HMI_Test_DB"   // DB46
// stored: InstanceOfName HMI_Test, InstanceOfType FB
"HMI_Test"
BEGIN
END_DATA_BLOCK

DATA_BLOCK "Oil_DB"   // DB40
// stored: InstanceOfName Oil, InstanceOfType FB
"Oil"
BEGIN
END_DATA_BLOCK

DATA_BLOCK "System_To_Moving_Pallets_DB"   // DB25
// stored: InstanceOfName System_To_Moving_Pallets, InstanceOfType FB
"System_To_Moving_Pallets"
BEGIN
END_DATA_BLOCK

DATA_BLOCK "Main_Safety_RTG1_DB"   // DB6, F_DB
NAME : FUSI
// stored: InstanceOfName Main_Safety_RTG1, InstanceOfType FB
"Main_Safety_RTG1"
BEGIN
END_DATA_BLOCK

DATA_BLOCK "Tippler_DB"   // DB400
// stored: AutoNumber false, InstanceOfName Tippler, InstanceOfType FB
"Tippler"
BEGIN
END_DATA_BLOCK

DATA_BLOCK "Side_Shifters_SS1"   // DB26
// stored: InstanceOfName Side_Shifters, InstanceOfType FB
"Side_Shifters"
BEGIN
END_DATA_BLOCK

DATA_BLOCK "Side_Shifters_SS2"   // DB17
// stored: InstanceOfName Side_Shifters, InstanceOfType FB
"Side_Shifters"
BEGIN
END_DATA_BLOCK

DATA_BLOCK "Timer_Buzzer_Column13_14"   // DB29
{ S7_Optimized_Access := 'TRUE' }
// stored: InstanceOfName IEC_TIMER, OfSystemLibElement IEC_TIMER, OfSystemLibVersion 1.0
"IEC_TIMER"
   // VAR
   //    PT : Time;
   //    ET { ExternalWritable := 'False'} : Time;
   //    IN : Bool;
   //    Q { ExternalWritable := 'False'} : Bool;
   // END_VAR
BEGIN
END_DATA_BLOCK

DATA_BLOCK "Timer_Buzzer_Column14_08"   // DB30
{ S7_Optimized_Access := 'TRUE' }
// stored: InstanceOfName IEC_TIMER, OfSystemLibElement IEC_TIMER, OfSystemLibVersion 1.0
"IEC_TIMER"
   // VAR
   //    PT : Time;
   //    ET { ExternalWritable := 'False'} : Time;
   //    IN : Bool;
   //    Q { ExternalWritable := 'False'} : Bool;
   // END_VAR
BEGIN
END_DATA_BLOCK

DATA_BLOCK "InstAnalyzeTokens"   // DB4
{ DB_Accessible_From_OPC_UA := 'FALSE' }
AUTHOR : SIEMENS AG
VERSION : 3.0
// stored: DBAccessibleFromOPCUA false, InstanceOfName AnalyzeTokens, InstanceOfType FB
"AnalyzeTokens"
BEGIN
END_DATA_BLOCK

DATA_BLOCK "InstDeserializeRows"   // DB9
{ DB_Accessible_From_OPC_UA := 'FALSE' }
// stored: DBAccessibleFromOPCUA false, InstanceOfName DeserializeRows, InstanceOfType FB
"DeserializeRows"
BEGIN
END_DATA_BLOCK

DATA_BLOCK "InstLSql_Microsoft"   // DB1
{ DB_Accessible_From_OPC_UA := 'FALSE' }
AUTHOR : (department/personInCharge/contact)
FAMILY : (family)
// stored: AutoNumber false, DBAccessibleFromOPCUA false, InstanceOfName LSql_Microsoft, InstanceOfType FB
"LSql_Microsoft"
   // VAR_INPUT
   //    enable { ExternalAccessible := 'False'; ExternalVisible := 'False'; ExternalWritable := 'False'} : Bool;
   //    connectionSettings { ExternalAccessible := 'False'; ExternalVisible := 'False'; ExternalWritable := 'False'} : "LSql_typeConnectionSettings";
   //    command { ExternalAccessible := 'False'; ExternalVisible := 'False'; ExternalWritable := 'False'} : String;
   //    executeCommand { ExternalAccessible := 'False'; ExternalVisible := 'False'; ExternalWritable := 'False'} : Bool;
   // END_VAR
   // VAR_OUTPUT
   //    valid { ExternalWritable := 'False'} : Bool;
   //    busy { ExternalWritable := 'False'} : Bool;
   //    error { ExternalWritable := 'False'} : Bool;
   //    status { ExternalWritable := 'False'} : Word;
   //    diagnostics { ExternalWritable := 'False'} : "LSql_typeDiagnostics";
   //    dataReceived { ExternalWritable := 'False'} : Bool;
   //    tdsTelegramArrayLength { ExternalWritable := 'False'} : UDInt;
   // END_VAR
   // VAR_IN_OUT
   //    tdsTelegramArray : Array[*] of Byte;
   // END_VAR
   // VAR
   //    instTsend { ExternalAccessible := 'False'; ExternalVisible := 'False'; ExternalWritable := 'False'} : TSEND;
   //    instTcon { ExternalAccessible := 'False'; ExternalVisible := 'False'; ExternalWritable := 'False'} : TCON;
   //    instTrcv { ExternalAccessible := 'False'; ExternalVisible := 'False'; ExternalWritable := 'False'} : TRCV;
   //    instTdiscon { ExternalAccessible := 'False'; ExternalVisible := 'False'; ExternalWritable := 'False'} : TDISCON;
   //    statEnableOld { ExternalAccessible := 'False'; ExternalVisible := 'False'; ExternalWritable := 'False'} : Bool;
   //    statEnable { ExternalAccessible := 'False'; ExternalVisible := 'False'; ExternalWritable := 'False'} : Bool;
   //    statValid { ExternalAccessible := 'False'; ExternalVisible := 'False'; ExternalWritable := 'False'} : Bool;
   //    statBusy { ExternalAccessible := 'False'; ExternalVisible := 'False'; ExternalWritable := 'False'} : Bool;
   //    statError { ExternalAccessible := 'False'; ExternalVisible := 'False'; ExternalWritable := 'False'} : Bool;
   //    statErrorUserCleared { ExternalAccessible := 'False'; ExternalVisible := 'False'; ExternalWritable := 'False'} : Bool;
   //    statErrorAutoCleared { ExternalAccessible := 'False'; ExternalVisible := 'False'; ExternalWritable := 'False'} : Bool;
   //    statStatus { ExternalAccessible := 'False'; ExternalVisible := 'False'; ExternalWritable := 'False'} : Word;
   //    statSubfunctionStatus { ExternalAccessible := 'False'; ExternalVisible := 'False'; ExternalWritable := 'False'} : Word;
   //    statFBErrorState { ExternalAccessible := 'False'; ExternalVisible := 'False'; ExternalWritable := 'False'} : DInt;
   //    statFBState { ExternalAccessible := 'False'; ExternalVisible := 'False'; ExternalWritable := 'False'} : DInt;
   //    statDisablingCompleted { ExternalAccessible := 'False'; ExternalVisible := 'False'; ExternalWritable := 'False'} : Bool;
   //    statEmptyDiagnostics { ExternalAccessible := 'False'; ExternalVisible := 'False'; ExternalWritable := 'False'} : "LSql_typeDiagnostics";
   //    statReceivedBytes { ExternalAccessible := 'False'; ExternalVisible := 'False'; ExternalWritable := 'False'} : UDInt;
   //    statExecuteSqlBatchOld { ExternalAccessible := 'False'; ExternalVisible := 'False'; ExternalWritable := 'False'} : Bool;
   //    statSqlBatchData { ExternalAccessible := 'False'; ExternalVisible := 'False'; ExternalWritable := 'False'} : "LSql_typeSqlBatchData";
   //    statSqlBatch { ExternalAccessible := 'False'; ExternalVisible := 'False'; ExternalWritable := 'False'} : Array[0..2047] of Byte;
   //    statSqlBatchLen { ExternalAccessible := 'False'; ExternalVisible := 'False'; ExternalWritable := 'False'} : DInt;
   //    statWriter { ExternalAccessible := 'False'; ExternalVisible := 'False'; ExternalWritable := 'False'} : Int;
   //    statStatusSqlBatchIntToWord { ExternalAccessible := 'False'; ExternalVisible := 'False'; ExternalWritable := 'False'} : Word;
   //    statLoginData { ExternalAccessible := 'False'; ExternalVisible := 'False'; ExternalWritable := 'False'} : "LSql_typeLoginData";
   //    statLogin { ExternalAccessible := 'False'; ExternalVisible := 'False'; ExternalWritable := 'False'} : Array[0..2047] of Byte;
   //    statLoginLen { ExternalAccessible := 'False'; ExternalVisible := 'False'; ExternalWritable := 'False'} : DInt;
   //    statStatusLoginIntToWord { ExternalAccessible := 'False'; ExternalVisible := 'False'; ExternalWritable := 'False'} : Word;
   //    statStatusPreLoginIntToWord { ExternalAccessible := 'False'; ExternalVisible := 'False'; ExternalWritable := 'False'} : Word;
   //    statPreLogin { ExternalAccessible := 'False'; ExternalVisible := 'False'; ExternalWritable := 'False'} : Array[0..2047] of Byte;
   //    statPreLoginLen { ExternalAccessible := 'False'; ExternalVisible := 'False'; ExternalWritable := 'False'} : DInt;
   //    statPreLoginCache { ExternalAccessible := 'False'; ExternalVisible := 'False'; ExternalWritable := 'False'} : Array[0..2047] of Byte;
   //    statPreLoginData { ExternalAccessible := 'False'; ExternalVisible := 'False'; ExternalWritable := 'False'} : "LSql_typePreloginData";
   //    statErrorWriteData { ExternalAccessible := 'False'; ExternalVisible := 'False'; ExternalWritable := 'False'} : Bool;
   //    statWriteData { ExternalAccessible := 'False'; ExternalVisible := 'False'; ExternalWritable := 'False'} : Word;
   //    statTransmissionSqlCommand { ExternalAccessible := 'False'; ExternalVisible := 'False'; ExternalWritable := 'False'} : Bool;
   //    statTdsDataReceived { ExternalAccessible := 'False'; ExternalVisible := 'False'; ExternalWritable := 'False'} : Bool;
   //    statTdsTelegramBytesReceived { ExternalAccessible := 'False'; ExternalVisible := 'False'; ExternalWritable := 'False'} : UDInt;
   //    statTdsFragmBufferBytesFilled { ExternalAccessible := 'False'; ExternalVisible := 'False'; ExternalWritable := 'False'} : UDInt;
   //    statTdsFragmHeaderBytesFilled { ExternalAccessible := 'False'; ExternalVisible := 'False'; ExternalWritable := 'False'} : UDInt;
   //    statTdsFragmLengthFromHeader { ExternalAccessible := 'False'; ExternalVisible := 'False'; ExternalWritable := 'False'} : UDInt;
   //    statTdsTelegramLength { ExternalAccessible := 'False'; ExternalVisible := 'False'; ExternalWritable := 'False'} : UDInt;
   //    statTdsFragmStatus { ExternalAccessible := 'False'; ExternalVisible := 'False'; ExternalWritable := 'False'} : Byte;
   //    statTrcvBlockBufferArray { ExternalAccessible := 'False'; ExternalVisible := 'False'; ExternalWritable := 'False'} : Array[0..2047] of Byte;
   //    statTdsFragmHeaderBuffer { ExternalAccessible := 'False'; ExternalVisible := 'False'; ExternalWritable := 'False'} : Array[0..7] of Byte;
   //    statTdsTelegramContinuing { ExternalAccessible := 'False'; ExternalVisible := 'False'; ExternalWritable := 'False'} : Bool;
   //    statTdsTelegramArrayLowerBound { ExternalAccessible := 'False'; ExternalVisible := 'False'; ExternalWritable := 'False'} : DInt;
   //    statTdsTelegramArrayUpperBound { ExternalAccessible := 'False'; ExternalVisible := 'False'; ExternalWritable := 'False'} : DInt;
   // END_VAR
BEGIN
END_DATA_BLOCK

DATA_BLOCK "CC_HydraulicUnit"   // DB27, Motion_DB
// stored: InstanceOfName TO_SpeedAxis, OfSystemLibElement TO_SpeedAxis, OfSystemLibVersion 7.0
TO_SpeedAxis   // technology object, version 7.0
   // // inherited from TO_Axis
   // // inherited from TO_Object
   // VAR
   //    Velocity { ExternalWritable := 'False'} : LReal;
   //    Acceleration { ExternalWritable := 'False'} : LReal;
   //    ActualSpeed { ExternalWritable := 'False'} : LReal;
   //    VelocitySetpoint { ExternalWritable := 'False'} : LReal;
   //    Actor { S7_SetPoint := 'True'} : TO_Struct_Actor;
   //    TorqueLimiting { S7_SetPoint := 'True'} : TO_Struct_TorqueLimiting;
   //    LoadGear { S7_SetPoint := 'True'} : TO_Struct_LoadGear;
   //    DynamicLimits { S7_SetPoint := 'True'} : TO_Struct_DynamicLimits;
   //    DynamicDefaults { S7_SetPoint := 'True'} : TO_Struct_DynamicDefaults;
   //    Override { S7_SetPoint := 'True'} : TO_Struct_Override;
   //    Units { ExternalWritable := 'False'; S7_SetPoint := 'True'} : TO_Struct_Units;
   //    StatusDrive { ExternalWritable := 'False'; S7_SetPoint := 'True'} : TO_Struct_StatusDrive;
   //    StatusTorqueData { ExternalWritable := 'False'; S7_SetPoint := 'True'} : TO_Struct_StatusTorqueData;
   //    StatusMotionIn { ExternalWritable := 'False'; S7_SetPoint := 'True'} : TO_Struct_StatusMotionIn;
   //    StatusWord { ExternalWritable := 'False'} : DWord;
   //    StatusWord2 { ExternalWritable := 'False'} : DWord;
   //    ErrorWord { ExternalWritable := 'False'} : DWord;
   //    ErrorDetail { ExternalWritable := 'False'; S7_SetPoint := 'True'} : TO_Struct_ErrorDetail;
   //    WarningWord { ExternalWritable := 'False'} : DWord;
   //    ControlPanel { S7_SetPoint := 'True'} : TO_Struct_ControlPanel;
   //    InternalToTrace { S7_SetPoint := 'True'} : Array[1..4] of TO_Struct_Internal;
   //    VirtualAxis { ExternalWritable := 'False'; S7_SetPoint := 'True'} : TO_Struct_VirtualAxis;
   //    Simulation { S7_SetPoint := 'True'} : TO_Struct_AxisSimulation;
   // END_VAR
BEGIN
   Actor.Interface.AddressIn.RID := 16#2080708;
   Actor.Interface.AddressIn.AREA := 16#81;
   Actor.Interface.AddressIn.OFFSET := 2760;
   Actor.Interface.AddressOut.RID := 16#2080709;
   Actor.Interface.AddressOut.AREA := 16#82;
   Actor.Interface.AddressOut.OFFSET := 2752;
   Actor.DriveParameter.ReferenceSpeed := 1460.0;
   Actor.DriveParameter.MaxSpeed := 1750.0;
   Actor.DriveParameter.ReferenceTorque := 102.31;
   DynamicLimits.MaxVelocity := 1750.0;
   DynamicLimits.MaxAcceleration := 583.333333333333;
   DynamicLimits.MaxDeceleration := 583.333333333333;
   DynamicLimits.MaxJerk := 11666.6666666667;
   DynamicDefaults.Velocity := 1460.0;
   DynamicDefaults.Acceleration := 8.11111111111111;
   DynamicDefaults.Deceleration := 4.86666666666667;
   DynamicDefaults.Jerk := 162.222222222219;
   DynamicDefaults.EmergencyDeceleration := 583.333333333333;
   _Actor.Interface.Telegram := 1;
END_DATA_BLOCK

DATA_BLOCK "CC_Vibrating_Unit_1"   // DB33, Motion_DB
// stored: AutoNumber false, InstanceOfName TO_SpeedAxis, OfSystemLibElement TO_SpeedAxis, OfSystemLibVersion 7.0
TO_SpeedAxis   // technology object, version 7.0
   // // inherited from TO_Axis
   // // inherited from TO_Object
   // VAR
   //    Velocity { ExternalWritable := 'False'} : LReal;
   //    Acceleration { ExternalWritable := 'False'} : LReal;
   //    ActualSpeed { ExternalWritable := 'False'} : LReal;
   //    VelocitySetpoint { ExternalWritable := 'False'} : LReal;
   //    Actor { S7_SetPoint := 'True'} : TO_Struct_Actor;
   //    TorqueLimiting { S7_SetPoint := 'True'} : TO_Struct_TorqueLimiting;
   //    LoadGear { S7_SetPoint := 'True'} : TO_Struct_LoadGear;
   //    DynamicLimits { S7_SetPoint := 'True'} : TO_Struct_DynamicLimits;
   //    DynamicDefaults { S7_SetPoint := 'True'} : TO_Struct_DynamicDefaults;
   //    Override { S7_SetPoint := 'True'} : TO_Struct_Override;
   //    Units { ExternalWritable := 'False'; S7_SetPoint := 'True'} : TO_Struct_Units;
   //    StatusDrive { ExternalWritable := 'False'; S7_SetPoint := 'True'} : TO_Struct_StatusDrive;
   //    StatusTorqueData { ExternalWritable := 'False'; S7_SetPoint := 'True'} : TO_Struct_StatusTorqueData;
   //    StatusMotionIn { ExternalWritable := 'False'; S7_SetPoint := 'True'} : TO_Struct_StatusMotionIn;
   //    StatusWord { ExternalWritable := 'False'} : DWord;
   //    StatusWord2 { ExternalWritable := 'False'} : DWord;
   //    ErrorWord { ExternalWritable := 'False'} : DWord;
   //    ErrorDetail { ExternalWritable := 'False'; S7_SetPoint := 'True'} : TO_Struct_ErrorDetail;
   //    WarningWord { ExternalWritable := 'False'} : DWord;
   //    ControlPanel { S7_SetPoint := 'True'} : TO_Struct_ControlPanel;
   //    InternalToTrace { S7_SetPoint := 'True'} : Array[1..4] of TO_Struct_Internal;
   //    VirtualAxis { ExternalWritable := 'False'; S7_SetPoint := 'True'} : TO_Struct_VirtualAxis;
   //    Simulation { S7_SetPoint := 'True'} : TO_Struct_AxisSimulation;
   // END_VAR
BEGIN
   Actor.DataAdaption := 1;
   Actor.Interface.AddressIn.RID := 16#2080708;
   Actor.Interface.AddressIn.AREA := 16#81;
   Actor.Interface.AddressIn.OFFSET := 3568;
   Actor.Interface.AddressOut.RID := 16#2080709;
   Actor.Interface.AddressOut.AREA := 16#82;
   Actor.Interface.AddressOut.OFFSET := 3560;
   Actor.DriveParameter.ReferenceSpeed := 2840.0;
   Actor.DriveParameter.ReferenceTorque := 18.8296;
   DynamicLimits.MaxAcceleration := 1000.0;
   DynamicLimits.MaxDeceleration := 1000.0;
   DynamicLimits.MaxJerk := 20000.0;
   DynamicDefaults.Velocity := 3000.0;
   DynamicDefaults.Acceleration := 16.6666666666667;
   DynamicDefaults.Deceleration := 16.6666666666667;
   DynamicDefaults.Jerk := 333.333333333333;
   DynamicDefaults.EmergencyDeceleration := 1000.0;
   _Actor.Interface.Telegram := 1;
   _Actor.DataAdaptionOffline := True;
END_DATA_BLOCK

DATA_BLOCK "CC_Vibrating_Unit_2"   // DB34, Motion_DB
// stored: AutoNumber false, InstanceOfName TO_SpeedAxis, OfSystemLibElement TO_SpeedAxis, OfSystemLibVersion 7.0
TO_SpeedAxis   // technology object, version 7.0
   // // inherited from TO_Axis
   // // inherited from TO_Object
   // VAR
   //    Velocity { ExternalWritable := 'False'} : LReal;
   //    Acceleration { ExternalWritable := 'False'} : LReal;
   //    ActualSpeed { ExternalWritable := 'False'} : LReal;
   //    VelocitySetpoint { ExternalWritable := 'False'} : LReal;
   //    Actor { S7_SetPoint := 'True'} : TO_Struct_Actor;
   //    TorqueLimiting { S7_SetPoint := 'True'} : TO_Struct_TorqueLimiting;
   //    LoadGear { S7_SetPoint := 'True'} : TO_Struct_LoadGear;
   //    DynamicLimits { S7_SetPoint := 'True'} : TO_Struct_DynamicLimits;
   //    DynamicDefaults { S7_SetPoint := 'True'} : TO_Struct_DynamicDefaults;
   //    Override { S7_SetPoint := 'True'} : TO_Struct_Override;
   //    Units { ExternalWritable := 'False'; S7_SetPoint := 'True'} : TO_Struct_Units;
   //    StatusDrive { ExternalWritable := 'False'; S7_SetPoint := 'True'} : TO_Struct_StatusDrive;
   //    StatusTorqueData { ExternalWritable := 'False'; S7_SetPoint := 'True'} : TO_Struct_StatusTorqueData;
   //    StatusMotionIn { ExternalWritable := 'False'; S7_SetPoint := 'True'} : TO_Struct_StatusMotionIn;
   //    StatusWord { ExternalWritable := 'False'} : DWord;
   //    StatusWord2 { ExternalWritable := 'False'} : DWord;
   //    ErrorWord { ExternalWritable := 'False'} : DWord;
   //    ErrorDetail { ExternalWritable := 'False'; S7_SetPoint := 'True'} : TO_Struct_ErrorDetail;
   //    WarningWord { ExternalWritable := 'False'} : DWord;
   //    ControlPanel { S7_SetPoint := 'True'} : TO_Struct_ControlPanel;
   //    InternalToTrace { S7_SetPoint := 'True'} : Array[1..4] of TO_Struct_Internal;
   //    VirtualAxis { ExternalWritable := 'False'; S7_SetPoint := 'True'} : TO_Struct_VirtualAxis;
   //    Simulation { S7_SetPoint := 'True'} : TO_Struct_AxisSimulation;
   // END_VAR
BEGIN
   Actor.DataAdaption := 1;
   Actor.Interface.AddressIn.RID := 16#2080708;
   Actor.Interface.AddressIn.AREA := 16#81;
   Actor.Interface.AddressIn.OFFSET := 3960;
   Actor.Interface.AddressOut.RID := 16#2080709;
   Actor.Interface.AddressOut.AREA := 16#82;
   Actor.Interface.AddressOut.OFFSET := 3952;
   Actor.DriveParameter.ReferenceSpeed := 2840.0;
   Actor.DriveParameter.ReferenceTorque := 18.8296;
   DynamicLimits.MaxAcceleration := 1000.0;
   DynamicLimits.MaxDeceleration := 1000.0;
   DynamicLimits.MaxJerk := 20000.0;
   DynamicDefaults.Velocity := 3000.0;
   DynamicDefaults.Acceleration := 1000.0;
   DynamicDefaults.Deceleration := 1000.0;
   DynamicDefaults.Jerk := 20000.0;
   DynamicDefaults.EmergencyDeceleration := 1000.0;
   _Actor.Interface.Telegram := 1;
   _Actor.DataAdaptionOffline := True;
END_DATA_BLOCK

DATA_BLOCK "CC_Vibrating_Unit_3"   // DB35, Motion_DB
// stored: AutoNumber false, InstanceOfName TO_SpeedAxis, OfSystemLibElement TO_SpeedAxis, OfSystemLibVersion 7.0
TO_SpeedAxis   // technology object, version 7.0
   // // inherited from TO_Axis
   // // inherited from TO_Object
   // VAR
   //    Velocity { ExternalWritable := 'False'} : LReal;
   //    Acceleration { ExternalWritable := 'False'} : LReal;
   //    ActualSpeed { ExternalWritable := 'False'} : LReal;
   //    VelocitySetpoint { ExternalWritable := 'False'} : LReal;
   //    Actor { S7_SetPoint := 'True'} : TO_Struct_Actor;
   //    TorqueLimiting { S7_SetPoint := 'True'} : TO_Struct_TorqueLimiting;
   //    LoadGear { S7_SetPoint := 'True'} : TO_Struct_LoadGear;
   //    DynamicLimits { S7_SetPoint := 'True'} : TO_Struct_DynamicLimits;
   //    DynamicDefaults { S7_SetPoint := 'True'} : TO_Struct_DynamicDefaults;
   //    Override { S7_SetPoint := 'True'} : TO_Struct_Override;
   //    Units { ExternalWritable := 'False'; S7_SetPoint := 'True'} : TO_Struct_Units;
   //    StatusDrive { ExternalWritable := 'False'; S7_SetPoint := 'True'} : TO_Struct_StatusDrive;
   //    StatusTorqueData { ExternalWritable := 'False'; S7_SetPoint := 'True'} : TO_Struct_StatusTorqueData;
   //    StatusMotionIn { ExternalWritable := 'False'; S7_SetPoint := 'True'} : TO_Struct_StatusMotionIn;
   //    StatusWord { ExternalWritable := 'False'} : DWord;
   //    StatusWord2 { ExternalWritable := 'False'} : DWord;
   //    ErrorWord { ExternalWritable := 'False'} : DWord;
   //    ErrorDetail { ExternalWritable := 'False'; S7_SetPoint := 'True'} : TO_Struct_ErrorDetail;
   //    WarningWord { ExternalWritable := 'False'} : DWord;
   //    ControlPanel { S7_SetPoint := 'True'} : TO_Struct_ControlPanel;
   //    InternalToTrace { S7_SetPoint := 'True'} : Array[1..4] of TO_Struct_Internal;
   //    VirtualAxis { ExternalWritable := 'False'; S7_SetPoint := 'True'} : TO_Struct_VirtualAxis;
   //    Simulation { S7_SetPoint := 'True'} : TO_Struct_AxisSimulation;
   // END_VAR
BEGIN
   Actor.DataAdaption := 1;
   Actor.Interface.AddressIn.RID := 16#2080708;
   Actor.Interface.AddressIn.AREA := 16#81;
   Actor.Interface.AddressIn.OFFSET := 4352;
   Actor.Interface.AddressOut.RID := 16#2080709;
   Actor.Interface.AddressOut.AREA := 16#82;
   Actor.Interface.AddressOut.OFFSET := 4352;
   Actor.DriveParameter.ReferenceSpeed := 2840.0;
   Actor.DriveParameter.ReferenceTorque := 18.83;
   DynamicLimits.MaxAcceleration := 1000.0;
   DynamicLimits.MaxDeceleration := 1000.0;
   DynamicLimits.MaxJerk := 20000.0;
   DynamicDefaults.Velocity := 3000.0;
   DynamicDefaults.Acceleration := 1000.0;
   DynamicDefaults.Deceleration := 1000.0;
   DynamicDefaults.Jerk := 20000.0;
   DynamicDefaults.EmergencyDeceleration := 1000.0;
   _Actor.Interface.Telegram := 1;
   _Actor.DataAdaptionOffline := True;
END_DATA_BLOCK

